LIN {X -0.200,Y -532.074,Z 1046.256,A 0.000,B 0.000,C 90.000,E1 262.129} C_DIS
LIN {X -0.087,Y -530.457,Z 1046.248,A 0.000,B 0.000,C 90.000,E1 260.679} C_DIS
LIN {X 0.126,Y -528.622,Z 1046.239,A 0.000,B 0.000,C 90.000,E1 258.926} C_DIS
LIN {X 0.276,Y -527.082,Z 1046.231,A 0.000,B 0.000,C 90.000,E1 257.465} C_DIS
LIN {X 0.047,Y -524.579,Z 1046.218,A 0.000,B 0.000,C 90.000,E1 255.172} C_DIS
LIN {X 0.007,Y -522.754,Z 1046.208,A 0.000,B 0.000,C 90.000,E1 253.433} C_DIS
LIN {X -0.210,Y -521.218,Z 1046.200,A 0.000,B 0.000,C 90.000,E1 252.000} C_DIS
LIN {X 0.188,Y -519.499,Z 1046.192,A 0.000,B 0.000,C 90.000,E1 250.496} C_DIS
LIN {X 0.026,Y -516.944,Z 1046.180,A 0.000,B 0.000,C 90.000,E1 248.465} C_DIS
LIN {X 0.090,Y -515.507,Z 1046.174,A 0.000,B 0.000,C 90.000,E1 247.283} C_DIS
LIN {X 0.257,Y -513.432,Z 1046.166,A 0.000,B 0.000,C 90.000,E1 245.793} C_DIS
LIN {X 0.125,Y -511.151,Z 1046.157,A 0.000,B 0.000,C 90.000,E1 244.332} C_DIS
LIN {X -0.049,Y -508.765,Z 1046.149,A 0.000,B 0.000,C 90.000,E1 242.871} C_DIS
LIN {X 0.003,Y -507.243,Z 1046.144,A 0.000,B 0.000,C 90.000,E1 241.975} C_DIS
LIN {X 0.221,Y -504.607,Z 1046.136,A 0.000,B 0.000,C 90.000,E1 240.461} C_DIS
LIN {X 0.260,Y -501.301,Z 1046.126,A 0.000,B 0.000,C 90.000,E1 238.663} C_DIS
LIN {X -0.205,Y -497.939,Z 1046.116,A 0.000,B 0.000,C 90.000,E1 236.914} C_DIS
LIN {X 0.081,Y -495.545,Z 1046.109,A 0.000,B 0.000,C 90.000,E1 235.674} C_DIS
LIN {X -0.224,Y -492.350,Z 1046.101,A 0.000,B 0.000,C 90.000,E1 234.196} C_DIS
LIN {X 0.097,Y -488.848,Z 1046.093,A 0.000,B 0.000,C 90.000,E1 232.637} C_DIS
LIN {X 0.258,Y -485.274,Z 1046.084,A 0.000,B 0.000,C 90.000,E1 231.090} C_DIS
LIN {X -0.202,Y -481.123,Z 1046.074,A 0.000,B 0.000,C 90.000,E1 229.299} C_DIS
LIN {X 0.022,Y -476.578,Z 1046.062,A 0.000,B 0.000,C 90.000,E1 227.106} C_DIS
LIN {X -0.022,Y -472.784,Z 1046.051,A 0.000,B 0.000,C 90.000,E1 225.243} C_DIS
LIN {X -0.230,Y -469.527,Z 1046.043,A 0.000,B 0.000,C 90.000,E1 223.704} C_DIS
LIN {X 0.180,Y -466.400,Z 1046.034,A 0.000,B 0.000,C 90.000,E1 222.081} C_DIS
LIN {X -0.129,Y -463.145,Z 1046.025,A 0.000,B 0.000,C 90.000,E1 220.539} C_DIS
LIN {X 0.201,Y -459.845,Z 1046.016,A 0.000,B 0.000,C 90.000,E1 218.910} C_DIS
LIN {X 0.010,Y -454.371,Z 1046.002,A 0.000,B 0.000,C 90.000,E1 216.377} C_DIS
LIN {X 0.035,Y -449.739,Z 1045.990,A 0.000,B 0.000,C 90.000,E1 214.119} C_DIS
LIN {X 0.044,Y -446.432,Z 1045.981,A 0.000,B 0.000,C 90.000,E1 212.498} C_DIS
LIN {X -0.006,Y -442.795,Z 1045.972,A 0.000,B 0.000,C 90.000,E1 210.875} C_DIS
LIN {X 0.202,Y -439.874,Z 1045.964,A 0.000,B 0.000,C 90.000,E1 209.539} C_DIS
LIN {X 0.141,Y -436.975,Z 1045.957,A 0.000,B 0.000,C 90.000,E1 208.231} C_DIS
LIN {X -0.139,Y -432.660,Z 1045.946,A 0.000,B 0.000,C 90.000,E1 206.283} C_DIS
LIN {X 0.031,Y -426.395,Z 1045.929,A 0.000,B 0.000,C 90.000,E1 203.259} C_DIS
LIN {X 0.105,Y -421.444,Z 1045.914,A 0.000,B 0.000,C 90.000,E1 200.556} C_DIS
LIN {X 0.074,Y -416.360,Z 1045.896,A 0.000,B 0.000,C 90.000,E1 197.166} C_DIS
LIN {X -0.051,Y -414.517,Z 1045.884,A 0.000,B 0.000,C 90.000,E1 195.134} C_DIS
LIN {X -0.136,Y -413.982,Z 1045.878,A 0.000,B 0.000,C 90.000,E1 194.120} C_DIS
LIN {X 0.007,Y -413.995,Z 1045.874,A 0.000,B 0.000,C 90.000,E1 193.244} C_DIS
LIN {X 0.114,Y -414.394,Z 1045.871,A 0.000,B 0.000,C 90.000,E1 192.715} C_DIS
LIN {X -0.119,Y -415.327,Z 1045.867,A 0.000,B 0.000,C 90.000,E1 192.063} C_DIS
LIN {X -0.073,Y -416.099,Z 1045.865,A 0.000,B 0.000,C 90.000,E1 191.715} C_DIS
LIN {X 0.043,Y -417.689,Z 1045.862,A 0.000,B 0.000,C 90.000,E1 191.186} C_DIS
LIN {X 0.167,Y -419.693,Z 1045.859,A 0.000,B 0.000,C 90.000,E1 190.658} C_DIS
LIN {X -0.114,Y -423.246,Z 1045.856,A 0.000,B 0.000,C 90.000,E1 190.018} C_DIS
LIN {X 0.049,Y -427.287,Z 1045.852,A 0.000,B 0.000,C 90.000,E1 189.321} C_DIS
LIN {X -0.124,Y -442.017,Z 1045.840,A 0.000,B 0.000,C 90.000,E1 187.182} C_DIS
LIN {X -0.190,Y -447.901,Z 1045.835,A 0.000,B 0.000,C 90.000,E1 186.372} C_DIS
LIN {X 0.121,Y -457.250,Z 1045.828,A 0.000,B 0.000,C 90.000,E1 185.049} C_DIS
LIN {X -0.200,Y -464.000,Z 1045.823,A 0.000,B 0.000,C 90.000,E1 184.131} C_DIS
LIN {X -0.094,Y -469.384,Z 1045.818,A 0.000,B 0.000,C 90.000,E1 183.326} C_DIS
LIN {X 0.062,Y -474.699,Z 1045.814,A 0.000,B 0.000,C 90.000,E1 182.522} C_DIS
LIN {X 0.213,Y -482.614,Z 1045.807,A 0.000,B 0.000,C 90.000,E1 181.260} C_DIS
LIN {X 0.159,Y -488.424,Z 1045.802,A 0.000,B 0.000,C 90.000,E1 180.344} C_DIS
LIN {X 0.170,Y -494.090,Z 1045.797,A 0.000,B 0.000,C 90.000,E1 179.427} C_DIS
LIN {X -0.071,Y -500.502,Z 1045.791,A 0.000,B 0.000,C 90.000,E1 178.396} C_DIS
LIN {X -0.222,Y -506.659,Z 1045.785,A 0.000,B 0.000,C 90.000,E1 177.364} C_DIS
LIN {X -0.212,Y -516.817,Z 1045.775,A 0.000,B 0.000,C 90.000,E1 175.584} C_DIS
LIN {X -0.104,Y -522.664,Z 1045.770,A 0.000,B 0.000,C 90.000,E1 174.546} C_DIS
LIN {X -0.239,Y -530.864,Z 1045.762,A 0.000,B 0.000,C 90.000,E1 173.109} C_DIS
LIN {X -0.101,Y -538.759,Z 1045.754,A 0.000,B 0.000,C 90.000,E1 171.659} C_DIS
LIN {X 0.197,Y -546.551,Z 1045.746,A 0.000,B 0.000,C 90.000,E1 170.208} C_DIS
LIN {X 0.092,Y -554.249,Z 1045.738,A 0.000,B 0.000,C 90.000,E1 168.814} C_DIS
LIN {X -0.184,Y -560.837,Z 1045.731,A 0.000,B 0.000,C 90.000,E1 167.589} C_DIS
LIN {X -0.241,Y -567.323,Z 1045.724,A 0.000,B 0.000,C 90.000,E1 166.353} C_DIS
LIN {X -0.013,Y -570.746,Z 1045.720,A 0.000,B 0.000,C 90.000,E1 165.644} C_DIS
LIN {X -0.218,Y -576.029,Z 1045.714,A 0.000,B 0.000,C 90.000,E1 164.574} C_DIS
LIN {X 0.205,Y -581.233,Z 1045.708,A 0.000,B 0.000,C 90.000,E1 163.449} C_DIS
LIN {X -0.245,Y -586.060,Z 1045.702,A 0.000,B 0.000,C 90.000,E1 162.417} C_DIS
LIN {X 0.066,Y -589.465,Z 1045.698,A 0.000,B 0.000,C 90.000,E1 161.583} C_DIS
LIN {X -0.278,Y -593.772,Z 1045.692,A 0.000,B 0.000,C 90.000,E1 160.550} C_DIS
LIN {X 0.203,Y -597.859,Z 1045.686,A 0.000,B 0.000,C 90.000,E1 159.444} C_DIS
LIN {X 0.056,Y -600.780,Z 1045.682,A 0.000,B 0.000,C 90.000,E1 158.666} C_DIS
LIN {X 0.007,Y -605.255,Z 1045.674,A 0.000,B 0.000,C 90.000,E1 157.358} C_DIS
LIN {X 0.090,Y -608.594,Z 1045.668,A 0.000,B 0.000,C 90.000,E1 156.305} C_DIS
LIN {X -0.127,Y -612.508,Z 1045.661,A 0.000,B 0.000,C 90.000,E1 155.025} C_DIS
LIN {X 0.017,Y -616.093,Z 1045.654,A 0.000,B 0.000,C 90.000,E1 153.717} C_DIS
LIN {X 0.213,Y -619.459,Z 1045.647,A 0.000,B 0.000,C 90.000,E1 152.410} C_DIS
LIN {X 0.185,Y -622.066,Z 1045.641,A 0.000,B 0.000,C 90.000,E1 151.385} C_DIS
LIN {X -0.044,Y -626.476,Z 1045.631,A 0.000,B 0.000,C 90.000,E1 149.616} C_DIS
LIN {X 0.123,Y -630.005,Z 1045.623,A 0.000,B 0.000,C 90.000,E1 148.074} C_DIS
LIN {X 0.324,Y -632.332,Z 1045.617,A 0.000,B 0.000,C 90.000,E1 147.041} C_DIS
LIN {X 0.055,Y -635.173,Z 1045.610,A 0.000,B 0.000,C 90.000,E1 145.801} C_DIS
LIN {X 0.215,Y -638.537,Z 1045.602,A 0.000,B 0.000,C 90.000,E1 144.276} C_DIS
LIN {X -0.106,Y -641.339,Z 1045.595,A 0.000,B 0.000,C 90.000,E1 143.050} C_DIS
LIN {X -0.052,Y -645.284,Z 1045.585,A 0.000,B 0.000,C 90.000,E1 141.295} C_DIS
LIN {X -0.340,Y -648.601,Z 1045.577,A 0.000,B 0.000,C 90.000,E1 139.828} C_DIS
LIN {X -0.154,Y -651.921,Z 1045.568,A 0.000,B 0.000,C 90.000,E1 138.324} C_DIS
LIN {X 0.417,Y -657.092,Z 1045.556,A 0.000,B 0.000,C 90.000,E1 136.053} C_DIS
LIN {X 0.177,Y -664.235,Z 1045.541,A 0.000,B 0.000,C 90.000,E1 133.380} C_DIS
LIN {X 0.181,Y -668.183,Z 1045.533,A 0.000,B 0.000,C 90.000,E1 131.919} C_DIS
LIN {X 0.256,Y -671.593,Z 1045.526,A 0.000,B 0.000,C 90.000,E1 130.701} C_DIS
LIN {X -0.021,Y -676.228,Z 1045.517,A 0.000,B 0.000,C 90.000,E1 129.036} C_DIS
LIN {X -0.277,Y -678.775,Z 1045.512,A 0.000,B 0.000,C 90.000,E1 128.096} C_DIS
LIN {X 0.064,Y -681.852,Z 1045.505,A 0.000,B 0.000,C 90.000,E1 126.870} C_DIS
LIN {X -0.307,Y -686.102,Z 1045.496,A 0.000,B 0.000,C 90.000,E1 125.231} C_DIS
LIN {X -0.417,Y -690.339,Z 1045.486,A 0.000,B 0.000,C 90.000,E1 123.579} C_DIS
LIN {X 0.276,Y -693.178,Z 1045.480,A 0.000,B 0.000,C 90.000,E1 122.339} C_DIS
LIN {X 0.049,Y -695.917,Z 1045.473,A 0.000,B 0.000,C 90.000,E1 121.180} C_DIS
LIN {X 0.194,Y -697.440,Z 1045.469,A 0.000,B 0.000,C 90.000,E1 120.463} C_DIS
LIN {X 0.015,Y -699.086,Z 1045.464,A 0.000,B 0.000,C 90.000,E1 119.539} C_DIS
LIN {X 0.200,Y -700.101,Z 1045.460,A 0.000,B 0.000,C 90.000,E1 118.821} C_DIS
LIN {X -0.024,Y -701.693,Z 1045.453,A 0.000,B 0.000,C 90.000,E1 117.436} C_DIS
LIN {X -0.209,Y -702.998,Z 1045.446,A 0.000,B 0.000,C 90.000,E1 116.283} C_DIS
LIN {X -0.024,Y -703.814,Z 1045.441,A 0.000,B 0.000,C 90.000,E1 115.335} C_DIS
LIN {X -0.109,Y -704.204,Z 1045.437,A 0.000,B 0.000,C 90.000,E1 114.643} C_DIS
LIN {X 0.168,Y -704.031,Z 1045.434,A 0.000,B 0.000,C 90.000,E1 114.155} C_DIS
LIN {X -0.190,Y -703.680,Z 1045.433,A 0.000,B 0.000,C 90.000,E1 113.951} C_DIS
LIN {X 0.089,Y -702.567,Z 1045.430,A 0.000,B 0.000,C 90.000,E1 113.462} C_DIS
LIN {X -0.278,Y -701.385,Z 1045.429,A 0.000,B 0.000,C 90.000,E1 113.259} C_DIS
LIN {X -0.011,Y -698.386,Z 1045.427,A 0.000,B 0.000,C 90.000,E1 112.770} C_DIS
LIN {X 0.120,Y -697.192,Z 1045.426,A 0.000,B 0.000,C 90.000,E1 112.642} C_DIS
LIN {X 0.249,Y -695.337,Z 1045.425,A 0.000,B 0.000,C 90.000,E1 112.514} C_DIS
LIN {X -0.172,Y -688.457,Z 1045.423,A 0.000,B 0.000,C 90.000,E1 112.206} C_DIS
LIN {X 0.181,Y -686.259,Z 1045.423,A 0.000,B 0.000,C 90.000,E1 112.099} C_DIS
LIN {X 0.154,Y -682.920,Z 1045.422,A 0.000,B 0.000,C 90.000,E1 112.025} C_DIS
LIN {X 0.001,Y -675.996,Z 1045.422,A 0.000,B 0.000,C 90.000,E1 111.950} C_DIS
LIN {X -0.058,Y -610.637,Z 1045.422,A 0.000,B 0.000,C 90.000,E1 111.950} C_DIS
LIN {X 0.150,Y -604.476,Z 1045.421,A 0.000,B 0.000,C 90.000,E1 111.716} C_DIS
LIN {X 0.007,Y -598.087,Z 1045.419,A 0.000,B 0.000,C 90.000,E1 111.408} C_DIS
LIN {X -0.080,Y -592.488,Z 1045.417,A 0.000,B 0.000,C 90.000,E1 111.046} C_DIS
LIN {X -0.061,Y -576.610,Z 1045.410,A 0.000,B 0.000,C 90.000,E1 109.758} C_DIS
LIN {X 0.286,Y -570.579,Z 1045.407,A 0.000,B 0.000,C 90.000,E1 109.268} C_DIS
LIN {X -0.275,Y -568.981,Z 1045.407,A 0.000,B 0.000,C 90.000,E1 109.214} C_DIS
LIN {X -0.188,Y -560.664,Z 1045.404,A 0.000,B 0.000,C 90.000,E1 108.725} C_DIS
LIN {X -0.120,Y -554.210,Z 1045.402,A 0.000,B 0.000,C 90.000,E1 108.362} C_DIS
LIN {X 0.095,Y -549.849,Z 1045.400,A 0.000,B 0.000,C 90.000,E1 108.055} C_DIS
LIN {X 0.152,Y -548.856,Z 1045.400,A 0.000,B 0.000,C 90.000,E1 107.946} C_DIS
LIN {X 0.230,Y -547.887,Z 1045.399,A 0.000,B 0.000,C 90.000,E1 107.819} C_DIS
LIN {X 0.188,Y -547.874,Z 1045.399,A 0.000,B 0.000,C 90.000,E1 107.819} C_DIS
LIN {X 0.273,Y -547.436,Z 1045.397,A 0.000,B 0.000,C 90.000,E1 107.511} C_DIS
LIN {X -0.215,Y -547.637,Z 1045.394,A 0.000,B 0.000,C 90.000,E1 106.858} C_DIS
LIN {X -0.069,Y -548.307,Z 1045.387,A 0.000,B 0.000,C 90.000,E1 105.717} C_DIS
LIN {X 0.139,Y -549.314,Z 1045.378,A 0.000,B 0.000,C 90.000,E1 104.008} C_DIS
LIN {X -0.248,Y -551.520,Z 1045.362,A 0.000,B 0.000,C 90.000,E1 101.243} C_DIS
LIN {X 0.091,Y -554.167,Z 1045.348,A 0.000,B 0.000,C 90.000,E1 98.690} C_DIS
LIN {X 0.263,Y -556.428,Z 1045.338,A 0.000,B 0.000,C 90.000,E1 96.720} C_DIS
LIN {X 0.021,Y -557.372,Z 1045.333,A 0.000,B 0.000,C 90.000,E1 95.910} C_DIS
LIN {X -0.073,Y -558.612,Z 1045.325,A 0.000,B 0.000,C 90.000,E1 94.531} C_DIS
LIN {X 0.209,Y -559.234,Z 1045.321,A 0.000,B 0.000,C 90.000,E1 93.669} C_DIS
LIN {X 0.117,Y -560.028,Z 1045.313,A 0.000,B 0.000,C 90.000,E1 92.293} C_DIS
LIN {X -0.057,Y -560.523,Z 1045.307,A 0.000,B 0.000,C 90.000,E1 91.203} C_DIS
LIN {X -0.047,Y -561.123,Z 1045.297,A 0.000,B 0.000,C 90.000,E1 89.542} C_DIS
LIN {X 0.087,Y -561.716,Z 1045.287,A 0.000,B 0.000,C 90.000,E1 87.593} C_DIS
LIN {X 0.262,Y -562.424,Z 1045.276,A 0.000,B 0.000,C 90.000,E1 85.641} C_DIS
LIN {X 0.259,Y -562.824,Z 1045.268,A 0.000,B 0.000,C 90.000,E1 84.261} C_DIS
LIN {X -0.154,Y -563.234,Z 1045.259,A 0.000,B 0.000,C 90.000,E1 82.648} C_DIS
LIN {X -0.008,Y -563.977,Z 1045.245,A 0.000,B 0.000,C 90.000,E1 80.151} C_DIS
LIN {X 0.262,Y -565.056,Z 1045.232,A 0.000,B 0.000,C 90.000,E1 77.645} C_DIS
LIN {X 0.082,Y -566.274,Z 1045.219,A 0.000,B 0.000,C 90.000,E1 75.463} C_DIS
LIN {X -0.138,Y -568.069,Z 1045.206,A 0.000,B 0.000,C 90.000,E1 73.015} C_DIS
LIN {X 0.099,Y -569.400,Z 1045.197,A 0.000,B 0.000,C 90.000,E1 71.348} C_DIS
LIN {X -0.169,Y -570.571,Z 1045.189,A 0.000,B 0.000,C 90.000,E1 70.007} C_DIS
LIN {X -0.032,Y -571.345,Z 1045.183,A 0.000,B 0.000,C 90.000,E1 68.901} C_DIS
LIN {X -0.054,Y -572.361,Z 1045.175,A 0.000,B 0.000,C 90.000,E1 67.539} C_DIS
LIN {X 0.135,Y -573.580,Z 1045.165,A 0.000,B 0.000,C 90.000,E1 65.613} C_DIS
LIN {X -0.302,Y -574.435,Z 1045.156,A 0.000,B 0.000,C 90.000,E1 64.024} C_DIS
LIN {X 0.048,Y -575.261,Z 1045.146,A 0.000,B 0.000,C 90.000,E1 62.359} C_DIS
LIN {X 0.024,Y -576.087,Z 1045.136,A 0.000,B 0.000,C 90.000,E1 60.461} C_DIS
LIN {X -0.329,Y -576.869,Z 1045.127,A 0.000,B 0.000,C 90.000,E1 58.869} C_DIS
LIN {X 0.117,Y -577.427,Z 1045.118,A 0.000,B 0.000,C 90.000,E1 57.199} C_DIS
LIN {X -0.239,Y -577.784,Z 1045.110,A 0.000,B 0.000,C 90.000,E1 55.881} C_DIS
LIN {X 0.220,Y -578.048,Z 1045.103,A 0.000,B 0.000,C 90.000,E1 54.482} C_DIS
LIN {X 0.054,Y -578.175,Z 1045.097,A 0.000,B 0.000,C 90.000,E1 53.417} C_DIS
LIN {X -0.114,Y -578.127,Z 1045.091,A 0.000,B 0.000,C 90.000,E1 52.351} C_DIS
LIN {X 0.070,Y -577.884,Z 1045.085,A 0.000,B 0.000,C 90.000,E1 51.251} C_DIS
LIN {X -0.040,Y -577.314,Z 1045.077,A 0.000,B 0.000,C 90.000,E1 49.908} C_DIS
LIN {X -0.162,Y -576.592,Z 1045.070,A 0.000,B 0.000,C 90.000,E1 48.566} C_DIS
LIN {X -0.063,Y -575.880,Z 1045.064,A 0.000,B 0.000,C 90.000,E1 47.472} C_DIS
LIN {X 0.029,Y -575.014,Z 1045.058,A 0.000,B 0.000,C 90.000,E1 46.377} C_DIS
LIN {X -0.306,Y -573.795,Z 1045.052,A 0.000,B 0.000,C 90.000,E1 45.324} C_DIS
LIN {X 0.039,Y -572.701,Z 1045.047,A 0.000,B 0.000,C 90.000,E1 44.474} C_DIS
LIN {X 0.079,Y -571.027,Z 1045.041,A 0.000,B 0.000,C 90.000,E1 43.380} C_DIS
LIN {X 0.017,Y -569.627,Z 1045.036,A 0.000,B 0.000,C 90.000,E1 42.567} C_DIS
LIN {X -0.092,Y -568.048,Z 1045.032,A 0.000,B 0.000,C 90.000,E1 41.757} C_DIS
LIN {X 0.198,Y -566.255,Z 1045.027,A 0.000,B 0.000,C 90.000,E1 40.906} C_DIS
LIN {X -0.011,Y -565.016,Z 1045.024,A 0.000,B 0.000,C 90.000,E1 40.378} C_DIS
LIN {X -0.122,Y -562.791,Z 1045.020,A 0.000,B 0.000,C 90.000,E1 39.564} C_DIS
LIN {X 0.083,Y -561.274,Z 1045.017,A 0.000,B 0.000,C 90.000,E1 38.991} C_DIS
LIN {X -0.064,Y -558.586,Z 1045.012,A 0.000,B 0.000,C 90.000,E1 38.177} C_DIS
LIN {X -0.162,Y -554.661,Z 1045.006,A 0.000,B 0.000,C 90.000,E1 37.076} C_DIS
LIN {X -0.013,Y -552.442,Z 1045.003,A 0.000,B 0.000,C 90.000,E1 36.503} C_DIS
LIN {X -0.143,Y -548.738,Z 1044.998,A 0.000,B 0.000,C 90.000,E1 35.678} C_DIS
LIN {X -0.133,Y -544.187,Z 1044.993,A 0.000,B 0.000,C 90.000,E1 34.692} C_DIS
LIN {X -0.046,Y -539.818,Z 1044.988,A 0.000,B 0.000,C 90.000,E1 33.833} C_DIS
LIN {X -0.006,Y -534.438,Z 1044.982,A 0.000,B 0.000,C 90.000,E1 32.832} C_DIS
LIN {X 0.100,Y -527.592,Z 1044.976,A 0.000,B 0.000,C 90.000,E1 31.671} C_DIS
LIN {X -0.247,Y -523.884,Z 1044.973,A 0.000,B 0.000,C 90.000,E1 31.131} C_DIS
LIN {X -0.071,Y -518.983,Z 1044.969,A 0.000,B 0.000,C 90.000,E1 30.384} C_DIS
LIN {X -0.033,Y -514.771,Z 1044.966,A 0.000,B 0.000,C 90.000,E1 29.795} C_DIS
LIN {X 0.152,Y -511.416,Z 1044.963,A 0.000,B 0.000,C 90.000,E1 29.333} C_DIS
LIN {X 0.021,Y -504.457,Z 1044.958,A 0.000,B 0.000,C 90.000,E1 28.487} C_DIS
LIN {X 0.020,Y -499.282,Z 1044.955,A 0.000,B 0.000,C 90.000,E1 27.897} C_DIS
LIN {X 0.238,Y -491.048,Z 1044.950,A 0.000,B 0.000,C 90.000,E1 27.001} C_DIS
LIN {X 0.081,Y -484.067,Z 1044.946,A 0.000,B 0.000,C 90.000,E1 26.309} C_DIS
LIN {X 0.103,Y -474.008,Z 1044.941,A 0.000,B 0.000,C 90.000,E1 25.335} C_DIS
LIN {X 0.155,Y -463.659,Z 1044.936,A 0.000,B 0.000,C 90.000,E1 24.387} C_DIS
LIN {X -0.078,Y -453.086,Z 1044.931,A 0.000,B 0.000,C 90.000,E1 23.515} C_DIS
LIN {X 0.100,Y -429.481,Z 1044.919,A 0.000,B 0.000,C 90.000,E1 21.408} C_DIS
LIN {X -0.117,Y -417.985,Z 1044.913,A 0.000,B 0.000,C 90.000,E1 20.301} C_DIS
LIN {X -0.190,Y -406.782,Z 1044.906,A 0.000,B 0.000,C 90.000,E1 19.087} C_DIS
LIN {X -0.056,Y -400.031,Z 1044.901,A 0.000,B 0.000,C 90.000,E1 18.236} C_DIS
LIN {X 0.082,Y -396.246,Z 1044.898,A 0.000,B 0.000,C 90.000,E1 17.692} C_DIS
LIN {X 0.117,Y -395.210,Z 1044.897,A 0.000,B 0.000,C 90.000,E1 17.511} C_DIS
LIN {X -0.148,Y -392.499,Z 1044.894,A 0.000,B 0.000,C 90.000,E1 16.913} C_DIS
LIN {X -0.073,Y -391.496,Z 1044.891,A 0.000,B 0.000,C 90.000,E1 16.370} C_DIS
LIN {X 0.141,Y -391.410,Z 1044.887,A 0.000,B 0.000,C 90.000,E1 15.717} C_DIS
LIN {X 0.067,Y -392.262,Z 1044.882,A 0.000,B 0.000,C 90.000,E1 14.662} C_DIS
LIN {X -0.027,Y -398.877,Z 1044.854,A 0.000,B 0.000,C 90.000,E1 9.726} C_DIS
LIN {X 0.163,Y -406.120,Z 1044.833,A 0.000,B 0.000,C 90.000,E1 5.853} C_DIS
LIN {X 0.113,Y -409.107,Z 1044.825,A 0.000,B 0.000,C 90.000,E1 4.473} C_DIS
LIN {X 0.091,Y -411.905,Z 1044.818,A 0.000,B 0.000,C 90.000,E1 3.269} C_DIS
LIN {X 0.107,Y -413.904,Z 1044.815,A 0.000,B 0.000,C 90.000,E1 2.751} C_DIS
LIN {X 0.198,Y -414.700,Z 1044.815,A 0.000,B 0.000,C 90.000,E1 2.579} C_DIS
LIN {X -0.114,Y -418.010,Z 1044.812,A 0.000,B 0.000,C 90.000,E1 2.121} C_DIS
LIN {X 0.084,Y -421.155,Z 1044.810,A 0.000,B 0.000,C 90.000,E1 1.776} C_DIS
LIN {X -0.058,Y -422.789,Z 1044.809,A 0.000,B 0.000,C 90.000,E1 1.661} C_DIS
LIN {X -0.160,Y -436.414,Z 1044.804,A 0.000,B 0.000,C 90.000,E1 0.802} C_DIS
LIN {X -0.182,Y -453.799,Z 1044.798,A 0.000,B 0.000,C 90.000,E1 359.714} C_DIS
LIN {X 0.113,Y -472.035,Z 1044.792,A 0.000,B 0.000,C 90.000,E1 358.568} C_DIS
LIN {X -0.212,Y -486.861,Z 1044.787,A 0.000,B 0.000,C 90.000,E1 357.707} C_DIS
LIN {X 0.018,Y -496.616,Z 1044.784,A 0.000,B 0.000,C 90.000,E1 357.078} C_DIS
LIN {X -0.004,Y -504.469,Z 1044.781,A 0.000,B 0.000,C 90.000,E1 356.560} C_DIS
LIN {X 0.215,Y -510.656,Z 1044.779,A 0.000,B 0.000,C 90.000,E1 356.102} C_DIS
LIN {X -0.040,Y -516.687,Z 1044.776,A 0.000,B 0.000,C 90.000,E1 355.698} C_DIS
LIN {X -0.028,Y -525.260,Z 1044.772,A 0.000,B 0.000,C 90.000,E1 355.008} C_DIS
LIN {X 0.107,Y -532.364,Z 1044.769,A 0.000,B 0.000,C 90.000,E1 354.375} C_DIS
LIN {X -0.068,Y -539.086,Z 1044.765,A 0.000,B 0.000,C 90.000,E1 353.742} C_DIS
LIN {X 0.038,Y -545.438,Z 1044.761,A 0.000,B 0.000,C 90.000,E1 353.053} C_DIS
LIN {X 0.263,Y -550.224,Z 1044.758,A 0.000,B 0.000,C 90.000,E1 352.470} C_DIS
LIN {X -0.141,Y -554.661,Z 1044.755,A 0.000,B 0.000,C 90.000,E1 351.951} C_DIS
LIN {X -0.140,Y -559.523,Z 1044.751,A 0.000,B 0.000,C 90.000,E1 351.254} C_DIS
LIN {X -0.092,Y -563.883,Z 1044.748,A 0.000,B 0.000,C 90.000,E1 350.557} C_DIS
LIN {X -0.249,Y -568.647,Z 1044.743,A 0.000,B 0.000,C 90.000,E1 349.746} C_DIS
LIN {X 0.307,Y -573.054,Z 1044.738,A 0.000,B 0.000,C 90.000,E1 348.870} C_DIS
LIN {X -0.213,Y -577.031,Z 1044.734,A 0.000,B 0.000,C 90.000,E1 348.105} C_DIS
LIN {X -0.018,Y -580.092,Z 1044.730,A 0.000,B 0.000,C 90.000,E1 347.409} C_DIS
LIN {X -0.245,Y -584.740,Z 1044.724,A 0.000,B 0.000,C 90.000,E1 346.353} C_DIS
LIN {X -0.195,Y -586.901,Z 1044.721,A 0.000,B 0.000,C 90.000,E1 345.811} C_DIS
LIN {X -0.230,Y -593.200,Z 1044.712,A 0.000,B 0.000,C 90.000,E1 344.212} C_DIS
LIN {X -0.133,Y -597.210,Z 1044.706,A 0.000,B 0.000,C 90.000,E1 343.142} C_DIS
LIN {X -0.270,Y -600.019,Z 1044.702,A 0.000,B 0.000,C 90.000,E1 342.362} C_DIS
LIN {X -0.185,Y -604.459,Z 1044.695,A 0.000,B 0.000,C 90.000,E1 341.040} C_DIS
LIN {X -0.331,Y -607.595,Z 1044.689,A 0.000,B 0.000,C 90.000,E1 340.007} C_DIS
LIN {X -0.164,Y -609.914,Z 1044.684,A 0.000,B 0.000,C 90.000,E1 339.209} C_DIS
LIN {X 0.028,Y -611.979,Z 1044.680,A 0.000,B 0.000,C 90.000,E1 338.411} C_DIS
LIN {X 0.173,Y -615.272,Z 1044.673,A 0.000,B 0.000,C 90.000,E1 337.102} C_DIS
LIN {X -0.186,Y -618.259,Z 1044.666,A 0.000,B 0.000,C 90.000,E1 335.845} C_DIS
LIN {X 0.062,Y -620.816,Z 1044.659,A 0.000,B 0.000,C 90.000,E1 334.537} C_DIS
LIN {X 0.052,Y -622.599,Z 1044.653,A 0.000,B 0.000,C 90.000,E1 333.512} C_DIS
LIN {X 0.066,Y -624.247,Z 1044.647,A 0.000,B 0.000,C 90.000,E1 332.487} C_DIS
LIN {X 0.096,Y -625.731,Z 1044.642,A 0.000,B 0.000,C 90.000,E1 331.463} C_DIS
LIN {X -0.092,Y -627.317,Z 1044.635,A 0.000,B 0.000,C 90.000,E1 330.205} C_DIS
LIN {X 0.086,Y -628.782,Z 1044.626,A 0.000,B 0.000,C 90.000,E1 328.663} C_DIS
LIN {X -0.067,Y -629.591,Z 1044.620,A 0.000,B 0.000,C 90.000,E1 327.661} C_DIS
LIN {X -0.035,Y -630.303,Z 1044.612,A 0.000,B 0.000,C 90.000,E1 326.135} C_DIS
LIN {X 0.172,Y -630.499,Z 1044.606,A 0.000,B 0.000,C 90.000,E1 325.102} C_DIS
LIN {X -0.292,Y -630.575,Z 1044.598,A 0.000,B 0.000,C 90.000,E1 323.623} C_DIS
LIN {X 0.343,Y -630.566,Z 1044.587,A 0.000,B 0.000,C 90.000,E1 321.537} C_DIS
LIN {X -0.079,Y -630.692,Z 1044.581,A 0.000,B 0.000,C 90.000,E1 320.561} C_DIS
LIN {X 0.219,Y -630.855,Z 1044.573,A 0.000,B 0.000,C 90.000,E1 319.013} C_DIS
LIN {X -0.017,Y -630.814,Z 1044.564,A 0.000,B 0.000,C 90.000,E1 317.514} C_DIS
LIN {X 0.103,Y -631.007,Z 1044.554,A 0.000,B 0.000,C 90.000,E1 315.729} C_DIS
LIN {X 0.204,Y -631.189,Z 1044.544,A 0.000,B 0.000,C 90.000,E1 313.947} C_DIS
LIN {X -0.137,Y -631.350,Z 1044.534,A 0.000,B 0.000,C 90.000,E1 312.204} C_DIS
LIN {X -0.315,Y -631.315,Z 1044.526,A 0.000,B 0.000,C 90.000,E1 310.701} C_DIS
LIN {X 0.164,Y -631.342,Z 1044.520,A 0.000,B 0.000,C 90.000,E1 309.644} C_DIS
LIN {X -0.251,Y -631.259,Z 1044.515,A 0.000,B 0.000,C 90.000,E1 308.669} C_DIS
LIN {X 0.031,Y -631.204,Z 1044.505,A 0.000,B 0.000,C 90.000,E1 306.870} C_DIS
LIN {X -0.122,Y -631.192,Z 1044.502,A 0.000,B 0.000,C 90.000,E1 306.377} C_DIS
LIN {X 0.244,Y -631.294,Z 1044.501,A 0.000,B 0.000,C 90.000,E1 306.091} C_DIS
LIN {X -0.124,Y -632.078,Z 1044.482,A 0.000,B 0.000,C 90.000,E1 302.832} C_DIS
LIN {X -0.030,Y -632.871,Z 1044.473,A 0.000,B 0.000,C 90.000,E1 301.052} C_DIS
LIN {X 0.012,Y -634.193,Z 1044.461,A 0.000,B 0.000,C 90.000,E1 299.027} C_DIS
LIN {X -0.035,Y -635.105,Z 1044.454,A 0.000,B 0.000,C 90.000,E1 297.769} C_DIS
LIN {X 0.146,Y -635.734,Z 1044.449,A 0.000,B 0.000,C 90.000,E1 296.744} C_DIS
LIN {X 0.288,Y -636.117,Z 1044.444,A 0.000,B 0.000,C 90.000,E1 295.976} C_DIS
LIN {X -0.318,Y -636.187,Z 1044.438,A 0.000,B 0.000,C 90.000,E1 294.771} C_DIS
LIN {X -0.392,Y -635.957,Z 1044.432,A 0.000,B 0.000,C 90.000,E1 293.770} C_DIS
LIN {X 0.197,Y -635.086,Z 1044.423,A 0.000,B 0.000,C 90.000,E1 292.206} C_DIS
LIN {X -0.004,Y -634.887,Z 1044.422,A 0.000,B 0.000,C 90.000,E1 291.972} C_DIS
LIN {X 0.065,Y -634.107,Z 1044.419,A 0.000,B 0.000,C 90.000,E1 291.461} C_DIS
LIN {X -0.134,Y -633.676,Z 1044.418,A 0.000,B 0.000,C 90.000,E1 291.227} C_DIS
LIN {X -0.304,Y -632.059,Z 1044.415,A 0.000,B 0.000,C 90.000,E1 290.737} C_DIS
LIN {X -0.280,Y -630.964,Z 1044.414,A 0.000,B 0.000,C 90.000,E1 290.482} C_DIS
LIN {X 0.122,Y -628.028,Z 1044.411,A 0.000,B 0.000,C 90.000,E1 289.939} C_DIS
LIN {X -0.032,Y -623.121,Z 1044.408,A 0.000,B 0.000,C 90.000,E1 289.450} C_DIS
LIN {X 0.011,Y -621.560,Z 1044.407,A 0.000,B 0.000,C 90.000,E1 289.322} C_DIS
LIN {X 0.138,Y -615.029,Z 1044.405,A 0.000,B 0.000,C 90.000,E1 288.906} C_DIS
LIN {X -0.091,Y -613.041,Z 1044.405,A 0.000,B 0.000,C 90.000,E1 288.833} C_DIS
LIN {X 0.046,Y -607.375,Z 1044.403,A 0.000,B 0.000,C 90.000,E1 288.598} C_DIS
LIN {X 0.191,Y -603.694,Z 1044.402,A 0.000,B 0.000,C 90.000,E1 288.417} C_DIS
LIN {X -0.107,Y -597.924,Z 1044.401,A 0.000,B 0.000,C 90.000,E1 288.236} C_DIS
LIN {X -0.192,Y -594.648,Z 1044.401,A 0.000,B 0.000,C 90.000,E1 288.109} C_DIS
LIN {X -0.226,Y -585.329,Z 1044.399,A 0.000,B 0.000,C 90.000,E1 287.819} C_DIS
LIN {X -0.271,Y -578.675,Z 1044.398,A 0.000,B 0.000,C 90.000,E1 287.638} C_DIS
LIN {X 0.227,Y -566.900,Z 1044.396,A 0.000,B 0.000,C 90.000,E1 287.221} C_DIS
LIN {X 0.213,Y -558.710,Z 1044.394,A 0.000,B 0.000,C 90.000,E1 286.913} C_DIS
LIN {X 0.090,Y -553.768,Z 1044.393,A 0.000,B 0.000,C 90.000,E1 286.677} C_DIS
LIN {X 0.200,Y -552.023,Z 1044.392,A 0.000,B 0.000,C 90.000,E1 286.567} C_DIS
LIN {X 0.039,Y -550.106,Z 1044.391,A 0.000,B 0.000,C 90.000,E1 286.315} C_DIS
LIN {X -0.221,Y -549.058,Z 1044.389,A 0.000,B 0.000,C 90.000,E1 286.024} C_DIS
LIN {X -0.156,Y -548.237,Z 1044.386,A 0.000,B 0.000,C 90.000,E1 285.426} C_DIS
LIN {X 0.281,Y -547.552,Z 1044.381,A 0.000,B 0.000,C 90.000,E1 284.537} C_DIS
LIN {X 0.031,Y -547.134,Z 1044.376,A 0.000,B 0.000,C 90.000,E1 283.592} C_DIS
LIN {X 0.000,Y -547.134,Z 1044.376,A 0.000,B 0.000,C 90.000,E1 283.592} C_DIS
LIN {X -0.052,Y -547.497,Z 1044.375,A 0.000,B 0.000,C 90.000,E1 283.536} C_DIS
LIN {X -0.093,Y -585.817,Z 1044.375,A 0.000,B 0.000,C 90.000,E1 283.536} C_DIS
LIN {X 0.293,Y -587.216,Z 1044.375,A 0.000,B 0.000,C 90.000,E1 283.411} C_DIS
LIN {X 0.022,Y -589.821,Z 1044.374,A 0.000,B 0.000,C 90.000,E1 283.244} C_DIS
LIN {X 0.212,Y -592.128,Z 1044.372,A 0.000,B 0.000,C 90.000,E1 283.008} C_DIS
LIN {X 0.074,Y -592.701,Z 1044.371,A 0.000,B 0.000,C 90.000,E1 282.771} C_DIS
LIN {X 0.043,Y -592.729,Z 1044.368,A 0.000,B 0.000,C 90.000,E1 282.243} C_DIS
LIN {X 0.015,Y -591.728,Z 1044.365,A 0.000,B 0.000,C 90.000,E1 281.715} C_DIS
LIN {X -0.233,Y -589.460,Z 1044.361,A 0.000,B 0.000,C 90.000,E1 281.074} C_DIS
LIN {X -0.071,Y -586.865,Z 1044.359,A 0.000,B 0.000,C 90.000,E1 280.658} C_DIS
LIN {X -0.286,Y -585.571,Z 1044.359,A 0.000,B 0.000,C 90.000,E1 280.546} C_DIS
LIN {X 0.182,Y -583.744,Z 1044.358,A 0.000,B 0.000,C 90.000,E1 280.366} C_DIS
LIN {X -0.297,Y -581.323,Z 1044.357,A 0.000,B 0.000,C 90.000,E1 280.197} C_DIS
LIN {X -0.199,Y -580.267,Z 1044.356,A 0.000,B 0.000,C 90.000,E1 280.074} C_DIS
LIN {X -0.282,Y -578.638,Z 1044.355,A 0.000,B 0.000,C 90.000,E1 279.962} C_DIS
LIN {X 0.249,Y -578.442,Z 1044.355,A 0.000,B 0.000,C 90.000,E1 279.905} C_DIS
LIN {X 0.209,Y -572.472,Z 1044.355,A 0.000,B 0.000,C 90.000,E1 279.905} C_DIS
LIN {X 0.158,Y -572.093,Z 1044.355,A 0.000,B 0.000,C 90.000,E1 279.905} C_DIS
LIN {X 0.103,Y -544.908,Z 1044.355,A 0.000,B 0.000,C 90.000,E1 279.905} C_DIS
LIN {X -0.242,Y -543.004,Z 1044.343,A 0.000,B 0.000,C 90.000,E1 277.757} C_DIS
LIN {X 0.096,Y -541.398,Z 1044.330,A 0.000,B 0.000,C 90.000,E1 275.454} C_DIS
LIN {X -0.204,Y -540.168,Z 1044.319,A 0.000,B 0.000,C 90.000,E1 273.498} C_DIS
LIN {X -0.043,Y -539.041,Z 1044.308,A 0.000,B 0.000,C 90.000,E1 271.489} C_DIS
LIN {X 0.017,Y -538.376,Z 1044.302,A 0.000,B 0.000,C 90.000,E1 270.344} C_DIS
LIN {X 0.090,Y -537.262,Z 1044.292,A 0.000,B 0.000,C 90.000,E1 268.625} C_DIS
LIN {X 0.140,Y -536.257,Z 1044.285,A 0.000,B 0.000,C 90.000,E1 267.192} C_DIS
LIN {X 0.173,Y -535.448,Z 1044.278,A 0.000,B 0.000,C 90.000,E1 266.045} C_DIS
LIN {X 0.244,Y -534.002,Z 1044.267,A 0.000,B 0.000,C 90.000,E1 264.033} C_DIS
LIN {X -0.209,Y -532.825,Z 1044.259,A 0.000,B 0.000,C 90.000,E1 262.648} C_DIS
LIN {X -0.080,Y -531.273,Z 1044.251,A 0.000,B 0.000,C 90.000,E1 261.197} C_DIS
LIN {X 0.127,Y -528.746,Z 1044.238,A 0.000,B 0.000,C 90.000,E1 258.870} C_DIS
LIN {X -0.237,Y -527.209,Z 1044.230,A 0.000,B 0.000,C 90.000,E1 257.465} C_DIS
LIN {X 0.180,Y -524.703,Z 1044.217,A 0.000,B 0.000,C 90.000,E1 255.102} C_DIS
LIN {X 0.004,Y -522.871,Z 1044.208,A 0.000,B 0.000,C 90.000,E1 253.378} C_DIS
LIN {X -0.215,Y -521.332,Z 1044.200,A 0.000,B 0.000,C 90.000,E1 251.945} C_DIS
LIN {X -0.135,Y -519.592,Z 1044.192,A 0.000,B 0.000,C 90.000,E1 250.477} C_DIS
LIN {X 0.016,Y -517.044,Z 1044.180,A 0.000,B 0.000,C 90.000,E1 248.411} C_DIS
LIN {X 0.078,Y -515.613,Z 1044.174,A 0.000,B 0.000,C 90.000,E1 247.230} C_DIS
LIN {X -0.228,Y -513.529,Z 1044.165,A 0.000,B 0.000,C 90.000,E1 245.793} C_DIS
LIN {X 0.105,Y -511.237,Z 1044.157,A 0.000,B 0.000,C 90.000,E1 244.280} C_DIS
LIN {X -0.169,Y -509.341,Z 1044.151,A 0.000,B 0.000,C 90.000,E1 243.127} C_DIS
LIN {X -0.108,Y -507.878,Z 1044.146,A 0.000,B 0.000,C 90.000,E1 242.231} C_DIS
LIN {X -0.249,Y -504.666,Z 1044.136,A 0.000,B 0.000,C 90.000,E1 240.461} C_DIS
LIN {X -0.080,Y -501.940,Z 1044.127,A 0.000,B 0.000,C 90.000,E1 238.948} C_DIS
LIN {X 0.155,Y -498.584,Z 1044.117,A 0.000,B 0.000,C 90.000,E1 237.120} C_DIS
LIN {X 0.038,Y -496.223,Z 1044.111,A 0.000,B 0.000,C 90.000,E1 235.928} C_DIS
LIN {X 0.035,Y -494.301,Z 1044.106,A 0.000,B 0.000,C 90.000,E1 235.022} C_DIS
LIN {X 0.009,Y -492.349,Z 1044.101,A 0.000,B 0.000,C 90.000,E1 234.116} C_DIS
LIN {X -0.057,Y -488.832,Z 1044.092,A 0.000,B 0.000,C 90.000,E1 232.603} C_DIS
LIN {X -0.020,Y -485.988,Z 1044.085,A 0.000,B 0.000,C 90.000,E1 231.376} C_DIS
LIN {X -0.094,Y -481.792,Z 1044.075,A 0.000,B 0.000,C 90.000,E1 229.542} C_DIS
LIN {X -0.206,Y -477.221,Z 1044.063,A 0.000,B 0.000,C 90.000,E1 227.391} C_DIS
LIN {X 0.111,Y -473.413,Z 1044.053,A 0.000,B 0.000,C 90.000,E1 225.486} C_DIS
LIN {X -0.086,Y -470.119,Z 1044.044,A 0.000,B 0.000,C 90.000,E1 223.947} C_DIS
LIN {X -0.009,Y -467.006,Z 1044.035,A 0.000,B 0.000,C 90.000,E1 222.366} C_DIS
LIN {X 0.093,Y -463.081,Z 1044.025,A 0.000,B 0.000,C 90.000,E1 220.458} C_DIS
LIN {X -0.227,Y -459.801,Z 1044.016,A 0.000,B 0.000,C 90.000,E1 218.910} C_DIS
LIN {X 0.221,Y -454.253,Z 1044.002,A 0.000,B 0.000,C 90.000,E1 216.297} C_DIS
LIN {X -0.016,Y -449.650,Z 1043.989,A 0.000,B 0.000,C 90.000,E1 214.072} C_DIS
LIN {X -0.138,Y -446.331,Z 1043.980,A 0.000,B 0.000,C 90.000,E1 212.467} C_DIS
LIN {X 0.236,Y -441.945,Z 1043.969,A 0.000,B 0.000,C 90.000,E1 210.463} C_DIS
LIN {X -0.175,Y -439.009,Z 1043.962,A 0.000,B 0.000,C 90.000,E1 209.205} C_DIS
LIN {X 0.108,Y -436.780,Z 1043.957,A 0.000,B 0.000,C 90.000,E1 208.180} C_DIS
LIN {X -0.170,Y -432.438,Z 1043.946,A 0.000,B 0.000,C 90.000,E1 206.232} C_DIS
LIN {X 0.002,Y -426.143,Z 1043.929,A 0.000,B 0.000,C 90.000,E1 203.206} C_DIS
LIN {X 0.045,Y -421.732,Z 1043.916,A 0.000,B 0.000,C 90.000,E1 200.844} C_DIS
LIN {X -0.204,Y -415.533,Z 1043.893,A 0.000,B 0.000,C 90.000,E1 196.804} C_DIS
LIN {X 0.015,Y -413.920,Z 1043.884,A 0.000,B 0.000,C 90.000,E1 195.064} C_DIS
LIN {X -0.181,Y -413.375,Z 1043.878,A 0.000,B 0.000,C 90.000,E1 194.064} C_DIS
LIN {X 0.022,Y -413.139,Z 1043.872,A 0.000,B 0.000,C 90.000,E1 193.008} C_DIS
LIN {X 0.185,Y -413.688,Z 1043.869,A 0.000,B 0.000,C 90.000,E1 192.299} C_DIS
LIN {X -0.140,Y -414.715,Z 1043.865,A 0.000,B 0.000,C 90.000,E1 191.658} C_DIS
LIN {X -0.014,Y -415.545,Z 1043.863,A 0.000,B 0.000,C 90.000,E1 191.299} C_DIS
LIN {X 0.080,Y -418.033,Z 1043.859,A 0.000,B 0.000,C 90.000,E1 190.602} C_DIS
LIN {X 0.138,Y -419.435,Z 1043.857,A 0.000,B 0.000,C 90.000,E1 190.254} C_DIS
LIN {X 0.227,Y -424.691,Z 1043.852,A 0.000,B 0.000,C 90.000,E1 189.321} C_DIS
LIN {X -0.197,Y -439.313,Z 1043.840,A 0.000,B 0.000,C 90.000,E1 187.239} C_DIS
LIN {X -0.175,Y -447.663,Z 1043.834,A 0.000,B 0.000,C 90.000,E1 186.087} C_DIS
LIN {X 0.092,Y -457.232,Z 1043.827,A 0.000,B 0.000,C 90.000,E1 184.759} C_DIS
LIN {X 0.130,Y -462.954,Z 1043.822,A 0.000,B 0.000,C 90.000,E1 183.955} C_DIS
LIN {X -0.018,Y -470.516,Z 1043.816,A 0.000,B 0.000,C 90.000,E1 182.865} C_DIS
LIN {X 0.130,Y -475.760,Z 1043.812,A 0.000,B 0.000,C 90.000,E1 182.064} C_DIS
LIN {X -0.226,Y -481.673,Z 1043.807,A 0.000,B 0.000,C 90.000,E1 181.203} C_DIS
LIN {X 0.189,Y -487.556,Z 1043.801,A 0.000,B 0.000,C 90.000,E1 180.229} C_DIS
LIN {X -0.102,Y -494.182,Z 1043.796,A 0.000,B 0.000,C 90.000,E1 179.198} C_DIS
LIN {X -0.032,Y -499.807,Z 1043.791,A 0.000,B 0.000,C 90.000,E1 178.282} C_DIS
LIN {X -0.254,Y -507.629,Z 1043.783,A 0.000,B 0.000,C 90.000,E1 176.963} C_DIS
LIN {X -0.149,Y -516.149,Z 1043.775,A 0.000,B 0.000,C 90.000,E1 175.469} C_DIS
LIN {X 0.178,Y -522.855,Z 1043.768,A 0.000,B 0.000,C 90.000,E1 174.261} C_DIS
LIN {X 0.107,Y -531.093,Z 1043.760,A 0.000,B 0.000,C 90.000,E1 172.818} C_DIS
LIN {X -0.075,Y -538.224,Z 1043.753,A 0.000,B 0.000,C 90.000,E1 171.546} C_DIS
LIN {X -0.150,Y -545.273,Z 1043.746,A 0.000,B 0.000,C 90.000,E1 170.274} C_DIS
LIN {X -0.186,Y -553.003,Z 1043.738,A 0.000,B 0.000,C 90.000,E1 168.870} C_DIS
LIN {X 0.064,Y -559.673,Z 1043.731,A 0.000,B 0.000,C 90.000,E1 167.589} C_DIS
LIN {X -0.008,Y -566.191,Z 1043.724,A 0.000,B 0.000,C 90.000,E1 166.353} C_DIS
LIN {X -0.163,Y -571.009,Z 1043.719,A 0.000,B 0.000,C 90.000,E1 165.408} C_DIS
LIN {X 0.189,Y -576.329,Z 1043.713,A 0.000,B 0.000,C 90.000,E1 164.283} C_DIS
LIN {X 0.226,Y -581.544,Z 1043.707,A 0.000,B 0.000,C 90.000,E1 163.196} C_DIS
LIN {X 0.165,Y -586.342,Z 1043.701,A 0.000,B 0.000,C 90.000,E1 162.127} C_DIS
LIN {X -0.217,Y -590.833,Z 1043.695,A 0.000,B 0.000,C 90.000,E1 161.094} C_DIS
LIN {X 0.333,Y -594.042,Z 1043.690,A 0.000,B 0.000,C 90.000,E1 160.242} C_DIS
LIN {X 0.154,Y -597.132,Z 1043.686,A 0.000,B 0.000,C 90.000,E1 159.464} C_DIS
LIN {X -0.349,Y -600.052,Z 1043.682,A 0.000,B 0.000,C 90.000,E1 158.720} C_DIS
LIN {X 0.220,Y -603.703,Z 1043.676,A 0.000,B 0.000,C 90.000,E1 157.614} C_DIS
LIN {X -0.277,Y -607.133,Z 1043.670,A 0.000,B 0.000,C 90.000,E1 156.613} C_DIS
LIN {X 0.078,Y -610.351,Z 1043.664,A 0.000,B 0.000,C 90.000,E1 155.537} C_DIS
LIN {X -0.298,Y -612.687,Z 1043.660,A 0.000,B 0.000,C 90.000,E1 154.793} C_DIS
LIN {X 0.110,Y -616.230,Z 1043.653,A 0.000,B 0.000,C 90.000,E1 153.461} C_DIS
LIN {X 0.300,Y -620.257,Z 1043.644,A 0.000,B 0.000,C 90.000,E1 151.897} C_DIS
LIN {X -0.270,Y -623.383,Z 1043.637,A 0.000,B 0.000,C 90.000,E1 150.667} C_DIS
LIN {X 0.046,Y -625.961,Z 1043.631,A 0.000,B 0.000,C 90.000,E1 149.616} C_DIS
LIN {X 0.203,Y -629.562,Z 1043.623,A 0.000,B 0.000,C 90.000,E1 148.074} C_DIS
LIN {X 0.399,Y -631.875,Z 1043.617,A 0.000,B 0.000,C 90.000,E1 147.041} C_DIS
LIN {X 0.123,Y -634.761,Z 1043.610,A 0.000,B 0.000,C 90.000,E1 145.801} C_DIS
LIN {X 0.275,Y -638.147,Z 1043.602,A 0.000,B 0.000,C 90.000,E1 144.276} C_DIS
LIN {X 0.061,Y -640.414,Z 1043.596,A 0.000,B 0.000,C 90.000,E1 143.290} C_DIS
LIN {X -0.329,Y -643.800,Z 1043.588,A 0.000,B 0.000,C 90.000,E1 141.823} C_DIS
LIN {X -0.228,Y -647.767,Z 1043.578,A 0.000,B 0.000,C 90.000,E1 140.070} C_DIS
LIN {X -0.005,Y -649.955,Z 1043.573,A 0.000,B 0.000,C 90.000,E1 139.057} C_DIS
LIN {X 0.209,Y -653.282,Z 1043.564,A 0.000,B 0.000,C 90.000,E1 137.553} C_DIS
LIN {X 0.379,Y -658.060,Z 1043.553,A 0.000,B 0.000,C 90.000,E1 135.567} C_DIS
LIN {X 0.182,Y -664.693,Z 1043.540,A 0.000,B 0.000,C 90.000,E1 133.137} C_DIS
LIN {X -0.246,Y -670.771,Z 1043.528,A 0.000,B 0.000,C 90.000,E1 130.987} C_DIS
LIN {X -0.014,Y -676.097,Z 1043.517,A 0.000,B 0.000,C 90.000,E1 129.036} C_DIS
LIN {X 0.132,Y -678.078,Z 1043.513,A 0.000,B 0.000,C 90.000,E1 128.302} C_DIS
LIN {X 0.067,Y -681.727,Z 1043.505,A 0.000,B 0.000,C 90.000,E1 126.870} C_DIS
LIN {X -0.307,Y -685.982,Z 1043.496,A 0.000,B 0.000,C 90.000,E1 125.231} C_DIS
LIN {X -0.419,Y -690.261,Z 1043.486,A 0.000,B 0.000,C 90.000,E1 123.579} C_DIS
LIN {X 0.272,Y -693.081,Z 1043.480,A 0.000,B 0.000,C 90.000,E1 122.339} C_DIS
LIN {X 0.043,Y -695.841,Z 1043.473,A 0.000,B 0.000,C 90.000,E1 121.180} C_DIS
LIN {X 0.188,Y -697.345,Z 1043.469,A 0.000,B 0.000,C 90.000,E1 120.463} C_DIS
LIN {X 0.009,Y -698.989,Z 1043.464,A 0.000,B 0.000,C 90.000,E1 119.539} C_DIS
LIN {X 0.192,Y -700.000,Z 1043.460,A 0.000,B 0.000,C 90.000,E1 118.821} C_DIS
LIN {X -0.034,Y -701.617,Z 1043.453,A 0.000,B 0.000,C 90.000,E1 117.436} C_DIS
LIN {X -0.220,Y -702.918,Z 1043.446,A 0.000,B 0.000,C 90.000,E1 116.283} C_DIS
LIN {X -0.035,Y -703.752,Z 1043.441,A 0.000,B 0.000,C 90.000,E1 115.335} C_DIS
LIN {X -0.122,Y -704.145,Z 1043.437,A 0.000,B 0.000,C 90.000,E1 114.643} C_DIS
LIN {X 0.156,Y -703.991,Z 1043.434,A 0.000,B 0.000,C 90.000,E1 114.155} C_DIS
LIN {X -0.204,Y -703.646,Z 1043.433,A 0.000,B 0.000,C 90.000,E1 113.951} C_DIS
LIN {X 0.076,Y -702.556,Z 1043.430,A 0.000,B 0.000,C 90.000,E1 113.462} C_DIS
LIN {X -0.291,Y -701.382,Z 1043.429,A 0.000,B 0.000,C 90.000,E1 113.259} C_DIS
LIN {X -0.024,Y -698.402,Z 1043.427,A 0.000,B 0.000,C 90.000,E1 112.770} C_DIS
LIN {X 0.106,Y -697.206,Z 1043.426,A 0.000,B 0.000,C 90.000,E1 112.642} C_DIS
LIN {X 0.236,Y -695.366,Z 1043.425,A 0.000,B 0.000,C 90.000,E1 112.514} C_DIS
LIN {X -0.196,Y -688.571,Z 1043.423,A 0.000,B 0.000,C 90.000,E1 112.206} C_DIS
LIN {X 0.131,Y -686.317,Z 1043.423,A 0.000,B 0.000,C 90.000,E1 112.099} C_DIS
LIN {X 0.079,Y -682.927,Z 1043.422,A 0.000,B 0.000,C 90.000,E1 112.025} C_DIS
LIN {X -0.083,Y -675.848,Z 1043.422,A 0.000,B 0.000,C 90.000,E1 111.950} C_DIS
LIN {X -0.135,Y -610.889,Z 1043.422,A 0.000,B 0.000,C 90.000,E1 111.950} C_DIS
LIN {X 0.079,Y -604.650,Z 1043.421,A 0.000,B 0.000,C 90.000,E1 111.716} C_DIS
LIN {X -0.012,Y -598.303,Z 1043.419,A 0.000,B 0.000,C 90.000,E1 111.408} C_DIS
LIN {X 0.128,Y -595.614,Z 1043.418,A 0.000,B 0.000,C 90.000,E1 111.227} C_DIS
LIN {X 0.168,Y -591.272,Z 1043.416,A 0.000,B 0.000,C 90.000,E1 110.918} C_DIS
LIN {X 0.062,Y -576.250,Z 1043.410,A 0.000,B 0.000,C 90.000,E1 109.704} C_DIS
LIN {X -0.140,Y -570.141,Z 1043.407,A 0.000,B 0.000,C 90.000,E1 109.268} C_DIS
LIN {X 0.021,Y -563.425,Z 1043.405,A 0.000,B 0.000,C 90.000,E1 108.852} C_DIS
LIN {X 0.088,Y -553.805,Z 1043.402,A 0.000,B 0.000,C 90.000,E1 108.308} C_DIS
LIN {X 0.255,Y -549.435,Z 1043.400,A 0.000,B 0.000,C 90.000,E1 108.000} C_DIS
LIN {X 0.234,Y -547.935,Z 1043.399,A 0.000,B 0.000,C 90.000,E1 107.819} C_DIS
LIN {X 0.193,Y -547.907,Z 1043.399,A 0.000,B 0.000,C 90.000,E1 107.819} C_DIS
LIN {X -0.241,Y -547.483,Z 1043.398,A 0.000,B 0.000,C 90.000,E1 107.583} C_DIS
LIN {X -0.106,Y -547.589,Z 1043.394,A 0.000,B 0.000,C 90.000,E1 106.968} C_DIS
LIN {X -0.115,Y -548.252,Z 1043.388,A 0.000,B 0.000,C 90.000,E1 105.843} C_DIS
LIN {X 0.233,Y -549.246,Z 1043.379,A 0.000,B 0.000,C 90.000,E1 104.120} C_DIS
LIN {X -0.162,Y -551.668,Z 1043.361,A 0.000,B 0.000,C 90.000,E1 101.074} C_DIS
LIN {X 0.157,Y -554.040,Z 1043.349,A 0.000,B 0.000,C 90.000,E1 98.803} C_DIS
LIN {X -0.232,Y -556.278,Z 1043.338,A 0.000,B 0.000,C 90.000,E1 96.891} C_DIS
LIN {X 0.142,Y -557.526,Z 1043.332,A 0.000,B 0.000,C 90.000,E1 95.739} C_DIS
LIN {X 0.055,Y -558.702,Z 1043.324,A 0.000,B 0.000,C 90.000,E1 94.359} C_DIS
LIN {X -0.133,Y -559.486,Z 1043.318,A 0.000,B 0.000,C 90.000,E1 93.269} C_DIS
LIN {X -0.217,Y -560.223,Z 1043.310,A 0.000,B 0.000,C 90.000,E1 91.892} C_DIS
LIN {X 0.078,Y -560.556,Z 1043.306,A 0.000,B 0.000,C 90.000,E1 91.031} C_DIS
LIN {X 0.090,Y -561.139,Z 1043.297,A 0.000,B 0.000,C 90.000,E1 89.370} C_DIS
LIN {X 0.223,Y -561.738,Z 1043.286,A 0.000,B 0.000,C 90.000,E1 87.421} C_DIS
LIN {X -0.258,Y -562.354,Z 1043.277,A 0.000,B 0.000,C 90.000,E1 85.812} C_DIS
LIN {X -0.259,Y -562.768,Z 1043.269,A 0.000,B 0.000,C 90.000,E1 84.432} C_DIS
LIN {X 0.044,Y -563.228,Z 1043.258,A 0.000,B 0.000,C 90.000,E1 82.470} C_DIS
LIN {X 0.105,Y -563.991,Z 1043.245,A 0.000,B 0.000,C 90.000,E1 79.982} C_DIS
LIN {X -0.067,Y -565.073,Z 1043.231,A 0.000,B 0.000,C 90.000,E1 77.521} C_DIS
LIN {X 0.003,Y -566.182,Z 1043.220,A 0.000,B 0.000,C 90.000,E1 75.589} C_DIS
LIN {X -0.233,Y -567.928,Z 1043.206,A 0.000,B 0.000,C 90.000,E1 73.142} C_DIS
LIN {X -0.163,Y -569.042,Z 1043.199,A 0.000,B 0.000,C 90.000,E1 71.764} C_DIS
LIN {X -0.084,Y -570.434,Z 1043.190,A 0.000,B 0.000,C 90.000,E1 70.115} C_DIS
LIN {X 0.208,Y -571.389,Z 1043.182,A 0.000,B 0.000,C 90.000,E1 68.720} C_DIS
LIN {X 0.185,Y -572.384,Z 1043.174,A 0.000,B 0.000,C 90.000,E1 67.358} C_DIS
LIN {X 0.010,Y -573.409,Z 1043.165,A 0.000,B 0.000,C 90.000,E1 65.741} C_DIS
LIN {X 0.084,Y -574.292,Z 1043.156,A 0.000,B 0.000,C 90.000,E1 64.101} C_DIS
LIN {X -0.240,Y -575.235,Z 1043.146,A 0.000,B 0.000,C 90.000,E1 62.231} C_DIS
LIN {X -0.268,Y -576.023,Z 1043.135,A 0.000,B 0.000,C 90.000,E1 60.333} C_DIS
LIN {X 0.167,Y -576.764,Z 1043.126,A 0.000,B 0.000,C 90.000,E1 58.663} C_DIS
LIN {X -0.022,Y -577.261,Z 1043.119,A 0.000,B 0.000,C 90.000,E1 57.327} C_DIS
LIN {X 0.255,Y -577.666,Z 1043.109,A 0.000,B 0.000,C 90.000,E1 55.674} C_DIS
LIN {X 0.064,Y -577.930,Z 1043.100,A 0.000,B 0.000,C 90.000,E1 54.069} C_DIS
LIN {X -0.108,Y -577.992,Z 1043.094,A 0.000,B 0.000,C 90.000,E1 53.004} C_DIS
LIN {X -0.088,Y -577.908,Z 1043.090,A 0.000,B 0.000,C 90.000,E1 52.190} C_DIS
LIN {X -0.063,Y -577.712,Z 1043.085,A 0.000,B 0.000,C 90.000,E1 51.376} C_DIS
LIN {X -0.015,Y -577.007,Z 1043.076,A 0.000,B 0.000,C 90.000,E1 49.747} C_DIS
LIN {X 0.001,Y -576.115,Z 1043.067,A 0.000,B 0.000,C 90.000,E1 48.119} C_DIS
LIN {X 0.091,Y -575.282,Z 1043.061,A 0.000,B 0.000,C 90.000,E1 47.025} C_DIS
LIN {X 0.043,Y -574.550,Z 1043.057,A 0.000,B 0.000,C 90.000,E1 46.215} C_DIS
LIN {X -0.008,Y -573.631,Z 1043.052,A 0.000,B 0.000,C 90.000,E1 45.405} C_DIS
LIN {X -0.067,Y -572.533,Z 1043.048,A 0.000,B 0.000,C 90.000,E1 44.595} C_DIS
LIN {X -0.139,Y -571.279,Z 1043.043,A 0.000,B 0.000,C 90.000,E1 43.785} C_DIS
LIN {X -0.113,Y -569.443,Z 1043.037,A 0.000,B 0.000,C 90.000,E1 42.690} C_DIS
LIN {X 0.196,Y -567.875,Z 1043.033,A 0.000,B 0.000,C 90.000,E1 41.838} C_DIS
LIN {X -0.203,Y -565.407,Z 1043.026,A 0.000,B 0.000,C 90.000,E1 40.782} C_DIS
LIN {X -0.049,Y -564.086,Z 1043.023,A 0.000,B 0.000,C 90.000,E1 40.216} C_DIS
LIN {X -0.072,Y -561.069,Z 1043.017,A 0.000,B 0.000,C 90.000,E1 39.116} C_DIS
LIN {X 0.214,Y -558.397,Z 1043.013,A 0.000,B 0.000,C 90.000,E1 38.257} C_DIS
LIN {X 0.113,Y -554.429,Z 1043.007,A 0.000,B 0.000,C 90.000,E1 37.156} C_DIS
LIN {X 0.328,Y -551.022,Z 1043.002,A 0.000,B 0.000,C 90.000,E1 36.297} C_DIS
LIN {X -0.131,Y -547.886,Z 1042.998,A 0.000,B 0.000,C 90.000,E1 35.644} C_DIS
LIN {X 0.308,Y -543.207,Z 1042.993,A 0.000,B 0.000,C 90.000,E1 34.612} C_DIS
LIN {X 0.221,Y -539.588,Z 1042.989,A 0.000,B 0.000,C 90.000,E1 33.913} C_DIS
LIN {X -0.192,Y -534.232,Z 1042.983,A 0.000,B 0.000,C 90.000,E1 32.959} C_DIS
LIN {X 0.087,Y -529.982,Z 1042.979,A 0.000,B 0.000,C 90.000,E1 32.212} C_DIS
LIN {X -0.123,Y -525.562,Z 1042.975,A 0.000,B 0.000,C 90.000,E1 31.514} C_DIS
LIN {X 0.121,Y -522.728,Z 1042.973,A 0.000,B 0.000,C 90.000,E1 31.052} C_DIS
LIN {X 0.185,Y -518.770,Z 1042.969,A 0.000,B 0.000,C 90.000,E1 30.463} C_DIS
LIN {X 0.221,Y -514.578,Z 1042.966,A 0.000,B 0.000,C 90.000,E1 29.873} C_DIS
LIN {X -0.040,Y -511.286,Z 1042.964,A 0.000,B 0.000,C 90.000,E1 29.461} C_DIS
LIN {X -0.058,Y -506.526,Z 1042.960,A 0.000,B 0.000,C 90.000,E1 28.871} C_DIS
LIN {X 0.083,Y -501.712,Z 1042.957,A 0.000,B 0.000,C 90.000,E1 28.281} C_DIS
LIN {X -0.008,Y -495.018,Z 1042.953,A 0.000,B 0.000,C 90.000,E1 27.564} C_DIS
LIN {X 0.090,Y -486.763,Z 1042.948,A 0.000,B 0.000,C 90.000,E1 26.693} C_DIS
LIN {X -0.046,Y -475.285,Z 1042.942,A 0.000,B 0.000,C 90.000,E1 25.591} C_DIS
LIN {X -0.039,Y -464.967,Z 1042.937,A 0.000,B 0.000,C 90.000,E1 24.643} C_DIS
LIN {X 0.054,Y -454.361,Z 1042.932,A 0.000,B 0.000,C 90.000,E1 23.718} C_DIS
LIN {X -0.053,Y -430.494,Z 1042.920,A 0.000,B 0.000,C 90.000,E1 21.642} C_DIS
LIN {X 0.070,Y -418.781,Z 1042.914,A 0.000,B 0.000,C 90.000,E1 20.482} C_DIS
LIN {X 0.185,Y -406.155,Z 1042.906,A 0.000,B 0.000,C 90.000,E1 19.087} C_DIS
LIN {X -0.113,Y -400.764,Z 1042.903,A 0.000,B 0.000,C 90.000,E1 18.471} C_DIS
LIN {X -0.105,Y -396.845,Z 1042.900,A 0.000,B 0.000,C 90.000,E1 17.946} C_DIS
LIN {X 0.048,Y -394.141,Z 1042.897,A 0.000,B 0.000,C 90.000,E1 17.457} C_DIS
LIN {X 0.169,Y -392.172,Z 1042.894,A 0.000,B 0.000,C 90.000,E1 16.913} C_DIS
LIN {X 0.133,Y -391.383,Z 1042.891,A 0.000,B 0.000,C 90.000,E1 16.386} C_DIS
LIN {X 0.201,Y -391.355,Z 1042.888,A 0.000,B 0.000,C 90.000,E1 15.843} C_DIS
LIN {X -0.150,Y -392.202,Z 1042.882,A 0.000,B 0.000,C 90.000,E1 14.828} C_DIS
LIN {X 0.050,Y -398.759,Z 1042.855,A 0.000,B 0.000,C 90.000,E1 9.849} C_DIS
LIN {X -0.108,Y -405.154,Z 1042.835,A 0.000,B 0.000,C 90.000,E1 6.372} C_DIS
LIN {X -0.166,Y -408.891,Z 1042.826,A 0.000,B 0.000,C 90.000,E1 4.645} C_DIS
LIN {X -0.201,Y -412.009,Z 1042.818,A 0.000,B 0.000,C 90.000,E1 3.269} C_DIS
LIN {X -0.185,Y -413.946,Z 1042.815,A 0.000,B 0.000,C 90.000,E1 2.751} C_DIS
LIN {X -0.185,Y -414.836,Z 1042.814,A 0.000,B 0.000,C 90.000,E1 2.579} C_DIS
LIN {X -0.163,Y -418.194,Z 1042.811,A 0.000,B 0.000,C 90.000,E1 2.064} C_DIS
LIN {X 0.016,Y -421.386,Z 1042.810,A 0.000,B 0.000,C 90.000,E1 1.718} C_DIS
LIN {X 0.186,Y -423.185,Z 1042.809,A 0.000,B 0.000,C 90.000,E1 1.547} C_DIS
LIN {X 0.040,Y -438.702,Z 1042.803,A 0.000,B 0.000,C 90.000,E1 0.573} C_DIS
LIN {X -0.086,Y -454.572,Z 1042.798,A 0.000,B 0.000,C 90.000,E1 359.599} C_DIS
LIN {X 0.218,Y -472.797,Z 1042.792,A 0.000,B 0.000,C 90.000,E1 358.453} C_DIS
LIN {X -0.186,Y -485.939,Z 1042.787,A 0.000,B 0.000,C 90.000,E1 357.707} C_DIS
LIN {X 0.238,Y -497.249,Z 1042.783,A 0.000,B 0.000,C 90.000,E1 356.963} C_DIS
LIN {X 0.223,Y -505.077,Z 1042.780,A 0.000,B 0.000,C 90.000,E1 356.445} C_DIS
LIN {X 0.089,Y -515.877,Z 1042.776,A 0.000,B 0.000,C 90.000,E1 355.698} C_DIS
LIN {X 0.084,Y -524.619,Z 1042.772,A 0.000,B 0.000,C 90.000,E1 355.008} C_DIS
LIN {X -0.240,Y -531.740,Z 1042.769,A 0.000,B 0.000,C 90.000,E1 354.432} C_DIS
LIN {X 0.164,Y -538.519,Z 1042.765,A 0.000,B 0.000,C 90.000,E1 353.742} C_DIS
LIN {X -0.210,Y -544.872,Z 1042.762,A 0.000,B 0.000,C 90.000,E1 353.109} C_DIS
LIN {X -0.049,Y -549.772,Z 1042.759,A 0.000,B 0.000,C 90.000,E1 352.534} C_DIS
LIN {X -0.095,Y -555.280,Z 1042.755,A 0.000,B 0.000,C 90.000,E1 351.837} C_DIS
LIN {X 0.162,Y -559.218,Z 1042.752,A 0.000,B 0.000,C 90.000,E1 351.254} C_DIS
LIN {X 0.116,Y -563.640,Z 1042.748,A 0.000,B 0.000,C 90.000,E1 350.566} C_DIS
LIN {X 0.053,Y -568.443,Z 1042.743,A 0.000,B 0.000,C 90.000,E1 349.746} C_DIS
LIN {X 0.046,Y -572.924,Z 1042.739,A 0.000,B 0.000,C 90.000,E1 348.926} C_DIS
LIN {X -0.029,Y -576.965,Z 1042.734,A 0.000,B 0.000,C 90.000,E1 348.117} C_DIS
LIN {X 0.286,Y -580.065,Z 1042.730,A 0.000,B 0.000,C 90.000,E1 347.409} C_DIS
LIN {X 0.062,Y -584.710,Z 1042.724,A 0.000,B 0.000,C 90.000,E1 346.353} C_DIS
LIN {X -0.210,Y -587.962,Z 1042.720,A 0.000,B 0.000,C 90.000,E1 345.574} C_DIS
LIN {X 0.082,Y -593.254,Z 1042.712,A 0.000,B 0.000,C 90.000,E1 344.212} C_DIS
LIN {X 0.183,Y -597.281,Z 1042.707,A 0.000,B 0.000,C 90.000,E1 343.142} C_DIS
LIN {X 0.048,Y -600.144,Z 1042.702,A 0.000,B 0.000,C 90.000,E1 342.362} C_DIS
LIN {X 0.138,Y -604.609,Z 1042.695,A 0.000,B 0.000,C 90.000,E1 341.040} C_DIS
LIN {X -0.005,Y -607.813,Z 1042.689,A 0.000,B 0.000,C 90.000,E1 340.007} C_DIS
LIN {X 0.111,Y -610.839,Z 1042.683,A 0.000,B 0.000,C 90.000,E1 338.954} C_DIS
LIN {X 0.047,Y -613.578,Z 1042.677,A 0.000,B 0.000,C 90.000,E1 337.922} C_DIS
LIN {X -0.323,Y -616.174,Z 1042.672,A 0.000,B 0.000,C 90.000,E1 336.922} C_DIS
LIN {X -0.110,Y -619.125,Z 1042.665,A 0.000,B 0.000,C 90.000,E1 335.613} C_DIS
LIN {X -0.150,Y -621.618,Z 1042.657,A 0.000,B 0.000,C 90.000,E1 334.332} C_DIS
LIN {X -0.147,Y -623.019,Z 1042.653,A 0.000,B 0.000,C 90.000,E1 333.563} C_DIS
LIN {X -0.114,Y -625.073,Z 1042.646,A 0.000,B 0.000,C 90.000,E1 332.281} C_DIS
LIN {X -0.071,Y -626.539,Z 1042.640,A 0.000,B 0.000,C 90.000,E1 331.257} C_DIS
LIN {X -0.242,Y -628.126,Z 1042.633,A 0.000,B 0.000,C 90.000,E1 329.999} C_DIS
LIN {X -0.387,Y -629.347,Z 1042.626,A 0.000,B 0.000,C 90.000,E1 328.742} C_DIS
LIN {X -0.186,Y -630.352,Z 1042.619,A 0.000,B 0.000,C 90.000,E1 327.454} C_DIS
LIN {X 0.026,Y -631.009,Z 1042.612,A 0.000,B 0.000,C 90.000,E1 326.167} C_DIS
LIN {X 0.080,Y -631.271,Z 1042.605,A 0.000,B 0.000,C 90.000,E1 324.895} C_DIS
LIN {X -0.372,Y -631.359,Z 1042.597,A 0.000,B 0.000,C 90.000,E1 323.417} C_DIS
LIN {X -0.085,Y -631.449,Z 1042.587,A 0.000,B 0.000,C 90.000,E1 321.618} C_DIS
LIN {X -0.134,Y -631.597,Z 1042.580,A 0.000,B 0.000,C 90.000,E1 320.356} C_DIS
LIN {X -0.182,Y -631.801,Z 1042.573,A 0.000,B 0.000,C 90.000,E1 319.094} C_DIS
LIN {X 0.181,Y -631.845,Z 1042.566,A 0.000,B 0.000,C 90.000,E1 317.796} C_DIS
LIN {X -0.256,Y -632.050,Z 1042.554,A 0.000,B 0.000,C 90.000,E1 315.810} C_DIS
LIN {X -0.020,Y -632.267,Z 1042.546,A 0.000,B 0.000,C 90.000,E1 314.271} C_DIS
LIN {X -0.332,Y -632.530,Z 1042.536,A 0.000,B 0.000,C 90.000,E1 312.528} C_DIS
LIN {X -0.067,Y -632.601,Z 1042.528,A 0.000,B 0.000,C 90.000,E1 310.987} C_DIS
LIN {X -0.097,Y -632.647,Z 1042.521,A 0.000,B 0.000,C 90.000,E1 309.725} C_DIS
LIN {X -0.001,Y -632.620,Z 1042.515,A 0.000,B 0.000,C 90.000,E1 308.705} C_DIS
LIN {X -0.176,Y -632.556,Z 1042.505,A 0.000,B 0.000,C 90.000,E1 306.950} C_DIS
LIN {X 0.057,Y -632.586,Z 1042.502,A 0.000,B 0.000,C 90.000,E1 306.423} C_DIS
LIN {X -0.233,Y -632.696,Z 1042.497,A 0.000,B 0.000,C 90.000,E1 305.438} C_DIS
LIN {X 0.122,Y -633.630,Z 1042.481,A 0.000,B 0.000,C 90.000,E1 302.625} C_DIS
LIN {X 0.283,Y -634.612,Z 1042.470,A 0.000,B 0.000,C 90.000,E1 300.590} C_DIS
LIN {X 0.287,Y -635.704,Z 1042.462,A 0.000,B 0.000,C 90.000,E1 299.077} C_DIS
LIN {X 0.012,Y -636.824,Z 1042.453,A 0.000,B 0.000,C 90.000,E1 297.590} C_DIS
LIN {X -0.348,Y -637.514,Z 1042.448,A 0.000,B 0.000,C 90.000,E1 296.616} C_DIS
LIN {X -0.188,Y -637.822,Z 1042.444,A 0.000,B 0.000,C 90.000,E1 295.848} C_DIS
LIN {X -0.080,Y -637.972,Z 1042.441,A 0.000,B 0.000,C 90.000,E1 295.335} C_DIS
LIN {X -0.081,Y -637.934,Z 1042.434,A 0.000,B 0.000,C 90.000,E1 294.079} C_DIS
LIN {X -0.182,Y -637.575,Z 1042.430,A 0.000,B 0.000,C 90.000,E1 293.334} C_DIS
LIN {X -0.238,Y -637.171,Z 1042.424,A 0.000,B 0.000,C 90.000,E1 292.333} C_DIS
LIN {X -0.389,Y -636.615,Z 1042.421,A 0.000,B 0.000,C 90.000,E1 291.844} C_DIS
LIN {X 0.283,Y -635.805,Z 1042.418,A 0.000,B 0.000,C 90.000,E1 291.280} C_DIS
LIN {X 0.090,Y -635.261,Z 1042.417,A 0.000,B 0.000,C 90.000,E1 291.046} C_DIS
LIN {X -0.068,Y -633.618,Z 1042.414,A 0.000,B 0.000,C 90.000,E1 290.556} C_DIS
LIN {X -0.041,Y -632.286,Z 1042.413,A 0.000,B 0.000,C 90.000,E1 290.301} C_DIS
LIN {X -0.230,Y -629.874,Z 1042.411,A 0.000,B 0.000,C 90.000,E1 289.939} C_DIS
LIN {X -0.219,Y -627.538,Z 1042.409,A 0.000,B 0.000,C 90.000,E1 289.685} C_DIS
LIN {X 0.266,Y -623.545,Z 1042.407,A 0.000,B 0.000,C 90.000,E1 289.268} C_DIS
LIN {X 0.170,Y -616.692,Z 1042.405,A 0.000,B 0.000,C 90.000,E1 288.852} C_DIS
LIN {X -0.064,Y -614.983,Z 1042.404,A 0.000,B 0.000,C 90.000,E1 288.779} C_DIS
LIN {X -0.112,Y -605.741,Z 1042.402,A 0.000,B 0.000,C 90.000,E1 288.417} C_DIS
LIN {X 0.229,Y -595.066,Z 1042.400,A 0.000,B 0.000,C 90.000,E1 288.000} C_DIS
LIN {X 0.248,Y -589.528,Z 1042.399,A 0.000,B 0.000,C 90.000,E1 287.819} C_DIS
LIN {X 0.128,Y -573.799,Z 1042.396,A 0.000,B 0.000,C 90.000,E1 287.347} C_DIS
LIN {X -0.312,Y -563.915,Z 1042.395,A 0.000,B 0.000,C 90.000,E1 287.040} C_DIS
LIN {X 0.215,Y -558.157,Z 1042.393,A 0.000,B 0.000,C 90.000,E1 286.732} C_DIS
LIN {X -0.155,Y -554.167,Z 1042.392,A 0.000,B 0.000,C 90.000,E1 286.551} C_DIS
LIN {X 0.093,Y -552.627,Z 1042.391,A 0.000,B 0.000,C 90.000,E1 286.315} C_DIS
LIN {X -0.129,Y -551.858,Z 1042.390,A 0.000,B 0.000,C 90.000,E1 286.205} C_DIS
LIN {X -0.188,Y -550.420,Z 1042.388,A 0.000,B 0.000,C 90.000,E1 285.788} C_DIS
LIN {X 0.171,Y -549.431,Z 1042.385,A 0.000,B 0.000,C 90.000,E1 285.190} C_DIS
LIN {X -0.211,Y -549.003,Z 1042.382,A 0.000,B 0.000,C 90.000,E1 284.828} C_DIS
LIN {X 0.296,Y -588.864,Z 1042.382,A 0.000,B 0.000,C 90.000,E1 284.773} C_DIS
LIN {X 0.127,Y -589.495,Z 1042.382,A 0.000,B 0.000,C 90.000,E1 284.773} C_DIS
LIN {X -0.013,Y -591.791,Z 1042.381,A 0.000,B 0.000,C 90.000,E1 284.647} C_DIS
LIN {X -0.255,Y -594.373,Z 1042.380,A 0.000,B 0.000,C 90.000,E1 284.481} C_DIS
LIN {X -0.027,Y -596.553,Z 1042.379,A 0.000,B 0.000,C 90.000,E1 284.245} C_DIS
LIN {X -0.045,Y -597.505,Z 1042.378,A 0.000,B 0.000,C 90.000,E1 284.120} C_DIS
LIN {X 0.084,Y -599.640,Z 1042.376,A 0.000,B 0.000,C 90.000,E1 283.716} C_DIS
LIN {X 0.012,Y -600.332,Z 1042.376,A 0.000,B 0.000,C 90.000,E1 283.592} C_DIS
LIN {X -0.061,Y -600.873,Z 1042.375,A 0.000,B 0.000,C 90.000,E1 283.467} C_DIS
LIN {X 0.242,Y -601.574,Z 1042.373,A 0.000,B 0.000,C 90.000,E1 283.175} C_DIS
LIN {X 0.268,Y -602.469,Z 1042.370,A 0.000,B 0.000,C 90.000,E1 282.647} C_DIS
LIN {X 0.303,Y -602.728,Z 1042.368,A 0.000,B 0.000,C 90.000,E1 282.119} C_DIS
LIN {X 0.026,Y -602.511,Z 1042.366,A 0.000,B 0.000,C 90.000,E1 281.883} C_DIS
LIN {X 0.218,Y -602.126,Z 1042.365,A 0.000,B 0.000,C 90.000,E1 281.602} C_DIS
LIN {X -0.058,Y -601.535,Z 1042.363,A 0.000,B 0.000,C 90.000,E1 281.366} C_DIS
LIN {X -0.026,Y -599.520,Z 1042.360,A 0.000,B 0.000,C 90.000,E1 280.838} C_DIS
LIN {X -0.011,Y -596.440,Z 1042.357,A 0.000,B 0.000,C 90.000,E1 280.310} C_DIS
LIN {X -0.124,Y -592.629,Z 1042.354,A 0.000,B 0.000,C 90.000,E1 279.792} C_DIS
LIN {X -0.227,Y -591.235,Z 1042.354,A 0.000,B 0.000,C 90.000,E1 279.670} C_DIS
LIN {X 0.153,Y -589.632,Z 1042.353,A 0.000,B 0.000,C 90.000,E1 279.500} C_DIS
LIN {X 0.157,Y -586.240,Z 1042.351,A 0.000,B 0.000,C 90.000,E1 279.151} C_DIS
LIN {X 0.204,Y -584.679,Z 1042.350,A 0.000,B 0.000,C 90.000,E1 279.029} C_DIS
LIN {X 0.015,Y -576.820,Z 1042.348,A 0.000,B 0.000,C 90.000,E1 278.681} C_DIS
LIN {X -0.251,Y -570.290,Z 1042.348,A 0.000,B 0.000,C 90.000,E1 278.624} C_DIS
LIN {X 0.266,Y -544.283,Z 1042.348,A 0.000,B 0.000,C 90.000,E1 278.568} C_DIS
LIN {X -0.145,Y -543.695,Z 1042.344,A 0.000,B 0.000,C 90.000,E1 277.936} C_DIS
LIN {X -0.187,Y -543.692,Z 1042.344,A 0.000,B 0.000,C 90.000,E1 277.936} C_DIS
LIN {X -0.223,Y -544.175,Z 1042.343,A 0.000,B 0.000,C 90.000,E1 277.701} C_DIS
LIN {X -0.142,Y -543.823,Z 1042.341,A 0.000,B 0.000,C 90.000,E1 277.409} C_DIS
LIN {X -0.118,Y -543.007,Z 1042.340,A 0.000,B 0.000,C 90.000,E1 277.239} C_DIS
LIN {X -0.159,Y -543.001,Z 1042.340,A 0.000,B 0.000,C 90.000,E1 277.239} C_DIS
LIN {X 0.196,Y -541.383,Z 1042.328,A 0.000,B 0.000,C 90.000,E1 275.106} C_DIS
LIN {X -0.181,Y -540.500,Z 1042.321,A 0.000,B 0.000,C 90.000,E1 273.726} C_DIS
LIN {X -0.015,Y -539.371,Z 1042.310,A 0.000,B 0.000,C 90.000,E1 271.718} C_DIS
LIN {X 0.049,Y -538.745,Z 1042.303,A 0.000,B 0.000,C 90.000,E1 270.573} C_DIS
LIN {X 0.130,Y -537.626,Z 1042.294,A 0.000,B 0.000,C 90.000,E1 268.854} C_DIS
LIN {X 0.190,Y -536.595,Z 1042.286,A 0.000,B 0.000,C 90.000,E1 267.421} C_DIS
LIN {X 0.227,Y -535.595,Z 1042.278,A 0.000,B 0.000,C 90.000,E1 265.988} C_DIS
LIN {X -0.230,Y -534.148,Z 1042.267,A 0.000,B 0.000,C 90.000,E1 264.033} C_DIS
LIN {X -0.152,Y -532.963,Z 1042.259,A 0.000,B 0.000,C 90.000,E1 262.591} C_DIS
LIN {X -0.022,Y -531.424,Z 1042.251,A 0.000,B 0.000,C 90.000,E1 261.141} C_DIS
LIN {X 0.217,Y -528.598,Z 1042.236,A 0.000,B 0.000,C 90.000,E1 258.522} C_DIS
LIN {X -0.130,Y -526.716,Z 1042.227,A 0.000,B 0.000,C 90.000,E1 256.825} C_DIS
LIN {X 0.237,Y -524.844,Z 1042.217,A 0.000,B 0.000,C 90.000,E1 255.046} C_DIS
LIN {X 0.059,Y -522.991,Z 1042.207,A 0.000,B 0.000,C 90.000,E1 253.323} C_DIS
LIN {X -0.001,Y -521.429,Z 1042.199,A 0.000,B 0.000,C 90.000,E1 251.873} C_DIS
LIN {X -0.085,Y -519.673,Z 1042.191,A 0.000,B 0.000,C 90.000,E1 250.423} C_DIS
LIN {X 0.063,Y -517.156,Z 1042.180,A 0.000,B 0.000,C 90.000,E1 248.358} C_DIS
LIN {X 0.121,Y -515.703,Z 1042.173,A 0.000,B 0.000,C 90.000,E1 247.177} C_DIS
LIN {X -0.188,Y -513.638,Z 1042.165,A 0.000,B 0.000,C 90.000,E1 245.741} C_DIS
LIN {X 0.031,Y -511.797,Z 1042.159,A 0.000,B 0.000,C 90.000,E1 244.537} C_DIS
LIN {X 0.094,Y -509.417,Z 1042.150,A 0.000,B 0.000,C 90.000,E1 243.050} C_DIS
LIN {X 0.158,Y -507.947,Z 1042.145,A 0.000,B 0.000,C 90.000,E1 242.153} C_DIS
LIN {X 0.147,Y -505.288,Z 1042.137,A 0.000,B 0.000,C 90.000,E1 240.667} C_DIS
LIN {X 0.198,Y -502.014,Z 1042.127,A 0.000,B 0.000,C 90.000,E1 238.869} C_DIS
LIN {X -0.253,Y -498.667,Z 1042.117,A 0.000,B 0.000,C 90.000,E1 237.120} C_DIS
LIN {X 0.044,Y -496.292,Z 1042.110,A 0.000,B 0.000,C 90.000,E1 235.881} C_DIS
LIN {X -0.246,Y -493.070,Z 1042.102,A 0.000,B 0.000,C 90.000,E1 234.402} C_DIS
LIN {X 0.091,Y -489.586,Z 1042.094,A 0.000,B 0.000,C 90.000,E1 232.844} C_DIS
LIN {X -0.035,Y -485.974,Z 1042.085,A 0.000,B 0.000,C 90.000,E1 231.331} C_DIS
LIN {X 0.069,Y -482.482,Z 1042.077,A 0.000,B 0.000,C 90.000,E1 229.784} C_DIS
LIN {X 0.082,Y -477.198,Z 1042.063,A 0.000,B 0.000,C 90.000,E1 227.310} C_DIS
LIN {X 0.296,Y -474.014,Z 1042.054,A 0.000,B 0.000,C 90.000,E1 225.729} C_DIS
LIN {X 0.110,Y -470.771,Z 1042.046,A 0.000,B 0.000,C 90.000,E1 224.190} C_DIS
LIN {X -0.043,Y -466.969,Z 1042.035,A 0.000,B 0.000,C 90.000,E1 222.324} C_DIS
LIN {X 0.069,Y -463.065,Z 1042.025,A 0.000,B 0.000,C 90.000,E1 220.415} C_DIS
LIN {X 0.045,Y -459.744,Z 1042.016,A 0.000,B 0.000,C 90.000,E1 218.830} C_DIS
LIN {X 0.122,Y -454.920,Z 1042.003,A 0.000,B 0.000,C 90.000,E1 216.583} C_DIS
LIN {X 0.159,Y -450.242,Z 1041.991,A 0.000,B 0.000,C 90.000,E1 214.326} C_DIS
LIN {X -0.128,Y -446.206,Z 1041.980,A 0.000,B 0.000,C 90.000,E1 212.418} C_DIS
LIN {X -0.131,Y -441.862,Z 1041.969,A 0.000,B 0.000,C 90.000,E1 210.463} C_DIS
LIN {X -0.082,Y -437.434,Z 1041.958,A 0.000,B 0.000,C 90.000,E1 208.487} C_DIS
LIN {X -0.140,Y -431.558,Z 1041.944,A 0.000,B 0.000,C 90.000,E1 205.848} C_DIS
LIN {X -0.006,Y -425.262,Z 1041.927,A 0.000,B 0.000,C 90.000,E1 202.823} C_DIS
LIN {X -0.106,Y -422.099,Z 1041.917,A 0.000,B 0.000,C 90.000,E1 201.153} C_DIS
LIN {X -0.063,Y -415.141,Z 1041.893,A 0.000,B 0.000,C 90.000,E1 196.732} C_DIS
LIN {X 0.063,Y -413.081,Z 1041.882,A 0.000,B 0.000,C 90.000,E1 194.662} C_DIS
LIN {X 0.117,Y -412.293,Z 1041.872,A 0.000,B 0.000,C 90.000,E1 192.939} C_DIS
LIN {X 0.184,Y -412.586,Z 1041.868,A 0.000,B 0.000,C 90.000,E1 192.243} C_DIS
LIN {X -0.065,Y -413.453,Z 1041.864,A 0.000,B 0.000,C 90.000,E1 191.591} C_DIS
LIN {X -0.027,Y -414.165,Z 1041.862,A 0.000,B 0.000,C 90.000,E1 191.243} C_DIS
LIN {X 0.073,Y -415.087,Z 1041.861,A 0.000,B 0.000,C 90.000,E1 190.894} C_DIS
LIN {X -0.133,Y -418.344,Z 1041.856,A 0.000,B 0.000,C 90.000,E1 190.074} C_DIS
LIN {X 0.175,Y -422.661,Z 1041.852,A 0.000,B 0.000,C 90.000,E1 189.265} C_DIS
LIN {X 0.136,Y -432.929,Z 1041.843,A 0.000,B 0.000,C 90.000,E1 187.757} C_DIS
LIN {X 0.176,Y -446.027,Z 1041.833,A 0.000,B 0.000,C 90.000,E1 185.967} C_DIS
LIN {X -0.209,Y -451.866,Z 1041.829,A 0.000,B 0.000,C 90.000,E1 185.220} C_DIS
LIN {X -0.087,Y -458.945,Z 1041.824,A 0.000,B 0.000,C 90.000,E1 184.245} C_DIS
LIN {X -0.134,Y -463.515,Z 1041.820,A 0.000,B 0.000,C 90.000,E1 183.612} C_DIS
LIN {X 0.078,Y -470.066,Z 1041.815,A 0.000,B 0.000,C 90.000,E1 182.636} C_DIS
LIN {X 0.223,Y -475.423,Z 1041.810,A 0.000,B 0.000,C 90.000,E1 181.835} C_DIS
LIN {X 0.106,Y -479.288,Z 1041.807,A 0.000,B 0.000,C 90.000,E1 181.260} C_DIS
LIN {X -0.194,Y -480.382,Z 1041.806,A 0.000,B 0.000,C 90.000,E1 181.146} C_DIS
LIN {X -0.086,Y -487.206,Z 1041.800,A 0.000,B 0.000,C 90.000,E1 180.057} C_DIS
LIN {X 0.079,Y -493.961,Z 1041.794,A 0.000,B 0.000,C 90.000,E1 178.969} C_DIS
LIN {X 0.164,Y -499.624,Z 1041.789,A 0.000,B 0.000,C 90.000,E1 178.051} C_DIS
LIN {X 0.010,Y -507.470,Z 1041.782,A 0.000,B 0.000,C 90.000,E1 176.731} C_DIS
LIN {X -0.130,Y -515.180,Z 1041.775,A 0.000,B 0.000,C 90.000,E1 175.412} C_DIS
LIN {X 0.173,Y -523.601,Z 1041.766,A 0.000,B 0.000,C 90.000,E1 173.913} C_DIS
LIN {X 0.119,Y -531.839,Z 1041.758,A 0.000,B 0.000,C 90.000,E1 172.470} C_DIS
LIN {X 0.148,Y -538.197,Z 1041.752,A 0.000,B 0.000,C 90.000,E1 171.319} C_DIS
LIN {X -0.104,Y -544.493,Z 1041.746,A 0.000,B 0.000,C 90.000,E1 170.208} C_DIS
LIN {X -0.249,Y -552.259,Z 1041.738,A 0.000,B 0.000,C 90.000,E1 168.814} C_DIS
LIN {X 0.105,Y -558.965,Z 1041.731,A 0.000,B 0.000,C 90.000,E1 167.521} C_DIS
LIN {X 0.159,Y -564.813,Z 1041.725,A 0.000,B 0.000,C 90.000,E1 166.408} C_DIS
LIN {X -0.124,Y -570.375,Z 1041.719,A 0.000,B 0.000,C 90.000,E1 165.338} C_DIS
LIN {X 0.226,Y -575.772,Z 1041.713,A 0.000,B 0.000,C 90.000,E1 164.212} C_DIS
LIN {X 0.008,Y -581.607,Z 1041.706,A 0.000,B 0.000,C 90.000,E1 163.015} C_DIS
LIN {X 0.203,Y -585.826,Z 1041.700,A 0.000,B 0.000,C 90.000,E1 162.054} C_DIS
LIN {X 0.186,Y -590.406,Z 1041.694,A 0.000,B 0.000,C 90.000,E1 160.986} C_DIS
LIN {X -0.261,Y -595.740,Z 1041.687,A 0.000,B 0.000,C 90.000,E1 159.699} C_DIS
LIN {X 0.250,Y -599.638,Z 1041.681,A 0.000,B 0.000,C 90.000,E1 158.592} C_DIS
LIN {X 0.260,Y -603.305,Z 1041.675,A 0.000,B 0.000,C 90.000,E1 157.539} C_DIS
LIN {X 0.265,Y -607.633,Z 1041.668,A 0.000,B 0.000,C 90.000,E1 156.230} C_DIS
LIN {X -0.177,Y -610.868,Z 1041.662,A 0.000,B 0.000,C 90.000,E1 155.229} C_DIS
LIN {X 0.233,Y -613.790,Z 1041.657,A 0.000,B 0.000,C 90.000,E1 154.152} C_DIS
LIN {X 0.113,Y -617.268,Z 1041.649,A 0.000,B 0.000,C 90.000,E1 152.871} C_DIS
LIN {X 0.053,Y -619.978,Z 1041.644,A 0.000,B 0.000,C 90.000,E1 151.847} C_DIS
LIN {X -0.226,Y -624.435,Z 1041.634,A 0.000,B 0.000,C 90.000,E1 150.078} C_DIS
LIN {X -0.092,Y -628.713,Z 1041.624,A 0.000,B 0.000,C 90.000,E1 148.280} C_DIS
LIN {X 0.089,Y -631.036,Z 1041.618,A 0.000,B 0.000,C 90.000,E1 147.248} C_DIS
LIN {X -0.202,Y -633.970,Z 1041.611,A 0.000,B 0.000,C 90.000,E1 146.008} C_DIS
LIN {X -0.067,Y -637.362,Z 1041.603,A 0.000,B 0.000,C 90.000,E1 144.482} C_DIS
LIN {X -0.290,Y -639.659,Z 1041.597,A 0.000,B 0.000,C 90.000,E1 143.497} C_DIS
LIN {X 0.221,Y -643.629,Z 1041.587,A 0.000,B 0.000,C 90.000,E1 141.698} C_DIS
LIN {X -0.185,Y -647.612,Z 1041.578,A 0.000,B 0.000,C 90.000,E1 139.989} C_DIS
LIN {X 0.039,Y -649.814,Z 1041.572,A 0.000,B 0.000,C 90.000,E1 138.976} C_DIS
LIN {X -0.182,Y -652.613,Z 1041.565,A 0.000,B 0.000,C 90.000,E1 137.757} C_DIS
LIN {X -0.008,Y -657.382,Z 1041.554,A 0.000,B 0.000,C 90.000,E1 135.769} C_DIS
LIN {X -0.231,Y -664.690,Z 1041.539,A 0.000,B 0.000,C 90.000,E1 133.095} C_DIS
LIN {X -0.209,Y -670.124,Z 1041.529,A 0.000,B 0.000,C 90.000,E1 131.148} C_DIS
LIN {X 0.420,Y -674.146,Z 1041.521,A 0.000,B 0.000,C 90.000,E1 129.644} C_DIS
LIN {X 0.140,Y -676.812,Z 1041.515,A 0.000,B 0.000,C 90.000,E1 128.705} C_DIS
LIN {X -0.234,Y -678.717,Z 1041.511,A 0.000,B 0.000,C 90.000,E1 128.016} C_DIS
LIN {X 0.103,Y -681.770,Z 1041.505,A 0.000,B 0.000,C 90.000,E1 126.790} C_DIS
LIN {X 0.289,Y -686.082,Z 1041.495,A 0.000,B 0.000,C 90.000,E1 125.105} C_DIS
LIN {X 0.188,Y -690.326,Z 1041.486,A 0.000,B 0.000,C 90.000,E1 123.452} C_DIS
LIN {X -0.058,Y -693.749,Z 1041.478,A 0.000,B 0.000,C 90.000,E1 122.054} C_DIS
LIN {X -0.045,Y -696.460,Z 1041.472,A 0.000,B 0.000,C 90.000,E1 120.875} C_DIS
LIN {X 0.117,Y -698.269,Z 1041.466,A 0.000,B 0.000,C 90.000,E1 119.922} C_DIS
LIN {X 0.291,Y -699.362,Z 1041.462,A 0.000,B 0.000,C 90.000,E1 119.205} C_DIS
LIN {X 0.131,Y -700.579,Z 1041.457,A 0.000,B 0.000,C 90.000,E1 118.281} C_DIS
LIN {X 0.207,Y -702.188,Z 1041.449,A 0.000,B 0.000,C 90.000,E1 116.873} C_DIS
LIN {X -0.245,Y -703.156,Z 1041.444,A 0.000,B 0.000,C 90.000,E1 115.976} C_DIS
LIN {X -0.053,Y -703.867,Z 1041.439,A 0.000,B 0.000,C 90.000,E1 115.027} C_DIS
LIN {X 0.230,Y -704.024,Z 1041.438,A 0.000,B 0.000,C 90.000,E1 114.771} C_DIS
LIN {X -0.135,Y -703.979,Z 1041.435,A 0.000,B 0.000,C 90.000,E1 114.335} C_DIS
LIN {X 0.148,Y -703.895,Z 1041.434,A 0.000,B 0.000,C 90.000,E1 114.079} C_DIS
LIN {X -0.216,Y -702.892,Z 1041.431,A 0.000,B 0.000,C 90.000,E1 113.643} C_DIS
LIN {X 0.062,Y -702.243,Z 1041.430,A 0.000,B 0.000,C 90.000,E1 113.387} C_DIS
LIN {X -0.179,Y -698.714,Z 1041.427,A 0.000,B 0.000,C 90.000,E1 112.823} C_DIS
LIN {X -0.048,Y -697.672,Z 1041.426,A 0.000,B 0.000,C 90.000,E1 112.695} C_DIS
LIN {X -0.186,Y -696.095,Z 1041.425,A 0.000,B 0.000,C 90.000,E1 112.589} C_DIS
LIN {X 0.048,Y -689.154,Z 1041.423,A 0.000,B 0.000,C 90.000,E1 112.206} C_DIS
LIN {X -0.270,Y -687.109,Z 1041.423,A 0.000,B 0.000,C 90.000,E1 112.153} C_DIS
LIN {X -0.153,Y -685.087,Z 1041.423,A 0.000,B 0.000,C 90.000,E1 112.078} C_DIS
LIN {X 0.093,Y -683.572,Z 1041.422,A 0.000,B 0.000,C 90.000,E1 112.025} C_DIS
LIN {X -0.170,Y -675.414,Z 1041.422,A 0.000,B 0.000,C 90.000,E1 111.950} C_DIS
LIN {X 0.365,Y -611.182,Z 1041.422,A 0.000,B 0.000,C 90.000,E1 111.897} C_DIS
LIN {X 0.119,Y -603.804,Z 1041.420,A 0.000,B 0.000,C 90.000,E1 111.663} C_DIS
LIN {X 0.050,Y -597.652,Z 1041.419,A 0.000,B 0.000,C 90.000,E1 111.354} C_DIS
LIN {X 0.104,Y -592.014,Z 1041.417,A 0.000,B 0.000,C 90.000,E1 110.972} C_DIS
LIN {X -0.145,Y -583.928,Z 1041.413,A 0.000,B 0.000,C 90.000,E1 110.355} C_DIS
LIN {X 0.309,Y -575.775,Z 1041.409,A 0.000,B 0.000,C 90.000,E1 109.631} C_DIS
LIN {X 0.018,Y -569.735,Z 1041.407,A 0.000,B 0.000,C 90.000,E1 109.214} C_DIS
LIN {X 0.053,Y -561.454,Z 1041.404,A 0.000,B 0.000,C 90.000,E1 108.725} C_DIS
LIN {X 0.112,Y -554.830,Z 1041.402,A 0.000,B 0.000,C 90.000,E1 108.362} C_DIS
LIN {X 0.234,Y -549.456,Z 1041.400,A 0.000,B 0.000,C 90.000,E1 108.000} C_DIS
LIN {X 0.192,Y -547.957,Z 1041.399,A 0.000,B 0.000,C 90.000,E1 107.819} C_DIS
LIN {X 0.150,Y -547.935,Z 1041.399,A 0.000,B 0.000,C 90.000,E1 107.819} C_DIS
LIN {X -0.242,Y -547.499,Z 1041.398,A 0.000,B 0.000,C 90.000,E1 107.583} C_DIS
LIN {X -0.110,Y -547.578,Z 1041.394,A 0.000,B 0.000,C 90.000,E1 106.985} C_DIS
LIN {X -0.054,Y -548.130,Z 1041.390,A 0.000,B 0.000,C 90.000,E1 106.134} C_DIS
LIN {X -0.145,Y -549.238,Z 1041.379,A 0.000,B 0.000,C 90.000,E1 104.175} C_DIS
LIN {X 0.110,Y -551.921,Z 1041.360,A 0.000,B 0.000,C 90.000,E1 100.782} C_DIS
LIN {X -0.114,Y -554.321,Z 1041.348,A 0.000,B 0.000,C 90.000,E1 98.568} C_DIS
LIN {X -0.076,Y -556.258,Z 1041.338,A 0.000,B 0.000,C 90.000,E1 96.891} C_DIS
LIN {X -0.258,Y -557.481,Z 1041.332,A 0.000,B 0.000,C 90.000,E1 95.796} C_DIS
LIN {X 0.133,Y -558.473,Z 1041.326,A 0.000,B 0.000,C 90.000,E1 94.645} C_DIS
LIN {X 0.022,Y -559.478,Z 1041.318,A 0.000,B 0.000,C 90.000,E1 93.269} C_DIS
LIN {X 0.047,Y -560.316,Z 1041.309,A 0.000,B 0.000,C 90.000,E1 91.604} C_DIS
LIN {X 0.051,Y -560.914,Z 1041.300,A 0.000,B 0.000,C 90.000,E1 89.943} C_DIS
LIN {X 0.067,Y -561.451,Z 1041.291,A 0.000,B 0.000,C 90.000,E1 88.282} C_DIS
LIN {X 0.006,Y -561.906,Z 1041.283,A 0.000,B 0.000,C 90.000,E1 86.906} C_DIS
LIN {X 0.080,Y -562.498,Z 1041.274,A 0.000,B 0.000,C 90.000,E1 85.241} C_DIS
LIN {X 0.129,Y -562.868,Z 1041.266,A 0.000,B 0.000,C 90.000,E1 83.856} C_DIS
LIN {X 0.030,Y -563.393,Z 1041.254,A 0.000,B 0.000,C 90.000,E1 81.659} C_DIS
LIN {X 0.190,Y -564.261,Z 1041.240,A 0.000,B 0.000,C 90.000,E1 79.162} C_DIS
LIN {X -0.134,Y -565.292,Z 1041.228,A 0.000,B 0.000,C 90.000,E1 76.992} C_DIS
LIN {X -0.089,Y -566.291,Z 1041.219,A 0.000,B 0.000,C 90.000,E1 75.338} C_DIS
LIN {X 0.077,Y -568.094,Z 1041.205,A 0.000,B 0.000,C 90.000,E1 72.851} C_DIS
LIN {X -0.016,Y -569.004,Z 1041.199,A 0.000,B 0.000,C 90.000,E1 71.764} C_DIS
LIN {X 0.061,Y -570.355,Z 1041.190,A 0.000,B 0.000,C 90.000,E1 70.115} C_DIS
LIN {X -0.001,Y -571.118,Z 1041.184,A 0.000,B 0.000,C 90.000,E1 69.028} C_DIS
LIN {X -0.030,Y -572.126,Z 1041.176,A 0.000,B 0.000,C 90.000,E1 67.667} C_DIS
LIN {X -0.208,Y -573.133,Z 1041.167,A 0.000,B 0.000,C 90.000,E1 66.049} C_DIS
LIN {X -0.133,Y -574.048,Z 1041.158,A 0.000,B 0.000,C 90.000,E1 64.409} C_DIS
LIN {X 0.053,Y -574.994,Z 1041.147,A 0.000,B 0.000,C 90.000,E1 62.487} C_DIS
LIN {X 0.178,Y -575.653,Z 1041.138,A 0.000,B 0.000,C 90.000,E1 60.845} C_DIS
LIN {X 0.159,Y -576.502,Z 1041.128,A 0.000,B 0.000,C 90.000,E1 58.948} C_DIS
LIN {X 0.107,Y -577.094,Z 1041.119,A 0.000,B 0.000,C 90.000,E1 57.327} C_DIS
LIN {X -0.252,Y -577.446,Z 1041.111,A 0.000,B 0.000,C 90.000,E1 56.008} C_DIS
LIN {X 0.047,Y -577.633,Z 1041.105,A 0.000,B 0.000,C 90.000,E1 54.895} C_DIS
LIN {X -0.123,Y -577.795,Z 1041.099,A 0.000,B 0.000,C 90.000,E1 53.829} C_DIS
LIN {X 0.170,Y -577.763,Z 1041.093,A 0.000,B 0.000,C 90.000,E1 52.718} C_DIS
LIN {X 0.030,Y -577.719,Z 1041.090,A 0.000,B 0.000,C 90.000,E1 52.190} C_DIS
LIN {X 0.053,Y -577.523,Z 1041.085,A 0.000,B 0.000,C 90.000,E1 51.376} C_DIS
LIN {X 0.096,Y -576.787,Z 1041.076,A 0.000,B 0.000,C 90.000,E1 49.747} C_DIS
LIN {X -0.034,Y -576.041,Z 1041.069,A 0.000,B 0.000,C 90.000,E1 48.405} C_DIS
LIN {X 0.060,Y -575.259,Z 1041.063,A 0.000,B 0.000,C 90.000,E1 47.310} C_DIS
LIN {X 0.014,Y -574.570,Z 1041.058,A 0.000,B 0.000,C 90.000,E1 46.500} C_DIS
LIN {X -0.023,Y -573.709,Z 1041.054,A 0.000,B 0.000,C 90.000,E1 45.688} C_DIS
LIN {X 0.027,Y -572.216,Z 1041.048,A 0.000,B 0.000,C 90.000,E1 44.595} C_DIS
LIN {X -0.048,Y -570.955,Z 1041.043,A 0.000,B 0.000,C 90.000,E1 43.785} C_DIS
LIN {X -0.026,Y -569.091,Z 1041.037,A 0.000,B 0.000,C 90.000,E1 42.690} C_DIS
LIN {X 0.278,Y -567.487,Z 1041.033,A 0.000,B 0.000,C 90.000,E1 41.838} C_DIS
LIN {X -0.236,Y -565.628,Z 1041.028,A 0.000,B 0.000,C 90.000,E1 41.067} C_DIS
LIN {X -0.018,Y -564.348,Z 1041.025,A 0.000,B 0.000,C 90.000,E1 40.496} C_DIS
LIN {X 0.229,Y -562.120,Z 1041.020,A 0.000,B 0.000,C 90.000,E1 39.644} C_DIS
LIN {X -0.006,Y -560.538,Z 1041.017,A 0.000,B 0.000,C 90.000,E1 39.116} C_DIS
LIN {X -0.165,Y -557.841,Z 1041.013,A 0.000,B 0.000,C 90.000,E1 38.302} C_DIS
LIN {X 0.007,Y -555.876,Z 1041.010,A 0.000,B 0.000,C 90.000,E1 37.729} C_DIS
LIN {X 0.238,Y -552.673,Z 1041.005,A 0.000,B 0.000,C 90.000,E1 36.870} C_DIS
LIN {X -0.071,Y -550.362,Z 1041.002,A 0.000,B 0.000,C 90.000,E1 36.343} C_DIS
LIN {X -0.092,Y -547.204,Z 1040.998,A 0.000,B 0.000,C 90.000,E1 35.644} C_DIS
LIN {X -0.281,Y -543.134,Z 1040.993,A 0.000,B 0.000,C 90.000,E1 34.818} C_DIS
LIN {X 0.243,Y -538.794,Z 1040.989,A 0.000,B 0.000,C 90.000,E1 33.913} C_DIS
LIN {X -0.180,Y -533.412,Z 1040.983,A 0.000,B 0.000,C 90.000,E1 32.959} C_DIS
LIN {X 0.092,Y -529.154,Z 1040.979,A 0.000,B 0.000,C 90.000,E1 32.212} C_DIS
LIN {X 0.004,Y -522.848,Z 1040.973,A 0.000,B 0.000,C 90.000,E1 31.209} C_DIS
LIN {X -0.164,Y -515.739,Z 1040.968,A 0.000,B 0.000,C 90.000,E1 30.207} C_DIS
LIN {X -0.067,Y -510.273,Z 1040.964,A 0.000,B 0.000,C 90.000,E1 29.461} C_DIS
LIN {X -0.091,Y -505.507,Z 1040.960,A 0.000,B 0.000,C 90.000,E1 28.871} C_DIS
LIN {X 0.037,Y -501.749,Z 1040.958,A 0.000,B 0.000,C 90.000,E1 28.409} C_DIS
LIN {X -0.095,Y -495.018,Z 1040.954,A 0.000,B 0.000,C 90.000,E1 27.692} C_DIS
LIN {X -0.220,Y -489.514,Z 1040.951,A 0.000,B 0.000,C 90.000,E1 27.129} C_DIS
LIN {X 0.092,Y -485.286,Z 1040.948,A 0.000,B 0.000,C 90.000,E1 26.668} C_DIS
LIN {X -0.111,Y -475.290,Z 1040.943,A 0.000,B 0.000,C 90.000,E1 25.720} C_DIS
LIN {X 0.013,Y -465.196,Z 1040.938,A 0.000,B 0.000,C 90.000,E1 24.771} C_DIS
LIN {X -0.226,Y -453.186,Z 1040.932,A 0.000,B 0.000,C 90.000,E1 23.770} C_DIS
LIN {X 0.024,Y -432.083,Z 1040.922,A 0.000,B 0.000,C 90.000,E1 21.897} C_DIS
LIN {X 0.086,Y -418.870,Z 1040.915,A 0.000,B 0.000,C 90.000,E1 20.610} C_DIS
LIN {X -0.119,Y -404.705,Z 1040.906,A 0.000,B 0.000,C 90.000,E1 19.087} C_DIS
LIN {X -0.158,Y -400.631,Z 1040.903,A 0.000,B 0.000,C 90.000,E1 18.598} C_DIS
LIN {X 0.031,Y -396.838,Z 1040.900,A 0.000,B 0.000,C 90.000,E1 18.055} C_DIS
LIN {X 0.028,Y -394.366,Z 1040.898,A 0.000,B 0.000,C 90.000,E1 17.638} C_DIS
LIN {X 0.138,Y -392.174,Z 1040.895,A 0.000,B 0.000,C 90.000,E1 17.040} C_DIS
LIN {X 0.054,Y -391.341,Z 1040.891,A 0.000,B 0.000,C 90.000,E1 16.386} C_DIS
LIN {X 0.123,Y -391.385,Z 1040.888,A 0.000,B 0.000,C 90.000,E1 15.843} C_DIS
LIN {X 0.151,Y -392.301,Z 1040.882,A 0.000,B 0.000,C 90.000,E1 14.773} C_DIS
LIN {X -0.002,Y -398.283,Z 1040.857,A 0.000,B 0.000,C 90.000,E1 10.197} C_DIS
LIN {X -0.178,Y -405.265,Z 1040.835,A 0.000,B 0.000,C 90.000,E1 6.372} C_DIS
LIN {X 0.171,Y -408.972,Z 1040.826,A 0.000,B 0.000,C 90.000,E1 4.588} C_DIS
LIN {X 0.142,Y -412.070,Z 1040.818,A 0.000,B 0.000,C 90.000,E1 3.212} C_DIS
LIN {X 0.159,Y -413.909,Z 1040.815,A 0.000,B 0.000,C 90.000,E1 2.694} C_DIS
LIN {X 0.158,Y -414.666,Z 1040.814,A 0.000,B 0.000,C 90.000,E1 2.522} C_DIS
LIN {X -0.185,Y -417.785,Z 1040.811,A 0.000,B 0.000,C 90.000,E1 2.064} C_DIS
LIN {X 0.022,Y -422.580,Z 1040.809,A 0.000,B 0.000,C 90.000,E1 1.547} C_DIS
LIN {X 0.212,Y -439.268,Z 1040.803,A 0.000,B 0.000,C 90.000,E1 0.458} C_DIS
LIN {X 0.119,Y -456.981,Z 1040.797,A 0.000,B 0.000,C 90.000,E1 359.370} C_DIS
LIN {X -0.111,Y -473.550,Z 1040.791,A 0.000,B 0.000,C 90.000,E1 358.396} C_DIS
LIN {X 0.088,Y -486.407,Z 1040.787,A 0.000,B 0.000,C 90.000,E1 357.593} C_DIS
LIN {X 0.023,Y -497.694,Z 1040.783,A 0.000,B 0.000,C 90.000,E1 356.906} C_DIS
LIN {X 0.194,Y -505.246,Z 1040.780,A 0.000,B 0.000,C 90.000,E1 356.388} C_DIS
LIN {X 0.057,Y -516.090,Z 1040.776,A 0.000,B 0.000,C 90.000,E1 355.641} C_DIS
LIN {X 0.019,Y -524.859,Z 1040.772,A 0.000,B 0.000,C 90.000,E1 354.951} C_DIS
LIN {X -0.250,Y -531.915,Z 1040.769,A 0.000,B 0.000,C 90.000,E1 354.375} C_DIS
LIN {X 0.190,Y -538.670,Z 1040.765,A 0.000,B 0.000,C 90.000,E1 353.685} C_DIS
LIN {X -0.139,Y -545.029,Z 1040.761,A 0.000,B 0.000,C 90.000,E1 353.053} C_DIS
LIN {X 0.044,Y -549.974,Z 1040.758,A 0.000,B 0.000,C 90.000,E1 352.470} C_DIS
LIN {X -0.072,Y -555.485,Z 1040.754,A 0.000,B 0.000,C 90.000,E1 351.781} C_DIS
LIN {X 0.184,Y -559.438,Z 1040.751,A 0.000,B 0.000,C 90.000,E1 351.197} C_DIS
LIN {X 0.232,Y -563.894,Z 1040.747,A 0.000,B 0.000,C 90.000,E1 350.500} C_DIS
LIN {X 0.077,Y -568.742,Z 1040.743,A 0.000,B 0.000,C 90.000,E1 349.690} C_DIS
LIN {X -0.167,Y -573.912,Z 1040.738,A 0.000,B 0.000,C 90.000,E1 348.757} C_DIS
LIN {X -0.118,Y -577.937,Z 1040.733,A 0.000,B 0.000,C 90.000,E1 347.937} C_DIS
LIN {X -0.132,Y -582.172,Z 1040.728,A 0.000,B 0.000,C 90.000,E1 346.992} C_DIS
LIN {X 0.239,Y -586.707,Z 1040.722,A 0.000,B 0.000,C 90.000,E1 345.880} C_DIS
LIN {X 0.247,Y -591.003,Z 1040.716,A 0.000,B 0.000,C 90.000,E1 344.810} C_DIS
LIN {X -0.255,Y -595.169,Z 1040.710,A 0.000,B 0.000,C 90.000,E1 343.795} C_DIS
LIN {X -0.133,Y -599.103,Z 1040.704,A 0.000,B 0.000,C 90.000,E1 342.725} C_DIS
LIN {X 0.222,Y -602.817,Z 1040.698,A 0.000,B 0.000,C 90.000,E1 341.638} C_DIS
LIN {X 0.140,Y -605.439,Z 1040.694,A 0.000,B 0.000,C 90.000,E1 340.859} C_DIS
LIN {X 0.008,Y -608.646,Z 1040.688,A 0.000,B 0.000,C 90.000,E1 339.826} C_DIS
LIN {X 0.134,Y -611.637,Z 1040.682,A 0.000,B 0.000,C 90.000,E1 338.773} C_DIS
LIN {X 0.078,Y -614.397,Z 1040.676,A 0.000,B 0.000,C 90.000,E1 337.741} C_DIS
LIN {X -0.283,Y -616.938,Z 1040.671,A 0.000,B 0.000,C 90.000,E1 336.741} C_DIS
LIN {X 0.209,Y -619.327,Z 1040.665,A 0.000,B 0.000,C 90.000,E1 335.665} C_DIS
LIN {X -0.080,Y -620.873,Z 1040.661,A 0.000,B 0.000,C 90.000,E1 334.921} C_DIS
LIN {X -0.089,Y -623.348,Z 1040.654,A 0.000,B 0.000,C 90.000,E1 333.640} C_DIS
LIN {X -0.046,Y -625.818,Z 1040.645,A 0.000,B 0.000,C 90.000,E1 332.103} C_DIS
LIN {X 0.304,Y -627.276,Z 1040.639,A 0.000,B 0.000,C 90.000,E1 331.051} C_DIS
LIN {X 0.150,Y -628.876,Z 1040.632,A 0.000,B 0.000,C 90.000,E1 329.793} C_DIS
LIN {X 0.020,Y -630.070,Z 1040.625,A 0.000,B 0.000,C 90.000,E1 328.535} C_DIS
LIN {X 0.235,Y -631.091,Z 1040.618,A 0.000,B 0.000,C 90.000,E1 327.248} C_DIS
LIN {X -0.063,Y -631.760,Z 1040.611,A 0.000,B 0.000,C 90.000,E1 326.008} C_DIS
LIN {X -0.353,Y -632.035,Z 1040.604,A 0.000,B 0.000,C 90.000,E1 324.769} C_DIS
LIN {X 0.088,Y -632.148,Z 1040.596,A 0.000,B 0.000,C 90.000,E1 323.210} C_DIS
LIN {X 0.023,Y -632.281,Z 1040.587,A 0.000,B 0.000,C 90.000,E1 321.698} C_DIS
LIN {X -0.014,Y -632.476,Z 1040.580,A 0.000,B 0.000,C 90.000,E1 320.436} C_DIS
LIN {X -0.050,Y -632.683,Z 1040.573,A 0.000,B 0.000,C 90.000,E1 319.175} C_DIS
LIN {X -0.142,Y -632.800,Z 1040.566,A 0.000,B 0.000,C 90.000,E1 317.919} C_DIS
LIN {X -0.087,Y -633.031,Z 1040.555,A 0.000,B 0.000,C 90.000,E1 315.891} C_DIS
LIN {X 0.170,Y -633.285,Z 1040.547,A 0.000,B 0.000,C 90.000,E1 314.352} C_DIS
LIN {X 0.097,Y -633.537,Z 1040.540,A 0.000,B 0.000,C 90.000,E1 313.095} C_DIS
LIN {X 0.136,Y -633.693,Z 1040.534,A 0.000,B 0.000,C 90.000,E1 312.081} C_DIS
LIN {X 0.060,Y -633.816,Z 1040.527,A 0.000,B 0.000,C 90.000,E1 310.825} C_DIS
LIN {X 0.162,Y -633.877,Z 1040.521,A 0.000,B 0.000,C 90.000,E1 309.806} C_DIS
LIN {X -0.218,Y -633.865,Z 1040.516,A 0.000,B 0.000,C 90.000,E1 308.830} C_DIS
LIN {X 0.135,Y -633.854,Z 1040.506,A 0.000,B 0.000,C 90.000,E1 307.030} C_DIS
LIN {X -0.267,Y -633.957,Z 1040.499,A 0.000,B 0.000,C 90.000,E1 305.804} C_DIS
LIN {X -0.041,Y -634.824,Z 1040.483,A 0.000,B 0.000,C 90.000,E1 303.007} C_DIS
LIN {X -0.187,Y -635.873,Z 1040.472,A 0.000,B 0.000,C 90.000,E1 301.003} C_DIS
LIN {X 0.257,Y -637.285,Z 1040.461,A 0.000,B 0.000,C 90.000,E1 298.949} C_DIS
LIN {X -0.042,Y -638.285,Z 1040.454,A 0.000,B 0.000,C 90.000,E1 297.719} C_DIS
LIN {X 0.188,Y -639.043,Z 1040.448,A 0.000,B 0.000,C 90.000,E1 296.693} C_DIS
LIN {X -0.206,Y -639.476,Z 1040.444,A 0.000,B 0.000,C 90.000,E1 295.976} C_DIS
LIN {X -0.028,Y -639.660,Z 1040.440,A 0.000,B 0.000,C 90.000,E1 295.207} C_DIS
LIN {X -0.059,Y -639.722,Z 1040.434,A 0.000,B 0.000,C 90.000,E1 294.207} C_DIS
LIN {X -0.142,Y -639.531,Z 1040.430,A 0.000,B 0.000,C 90.000,E1 293.462} C_DIS
LIN {X -0.170,Y -639.060,Z 1040.425,A 0.000,B 0.000,C 90.000,E1 292.461} C_DIS
LIN {X -0.259,Y -638.434,Z 1040.421,A 0.000,B 0.000,C 90.000,E1 291.716} C_DIS
LIN {X 0.195,Y -637.584,Z 1040.418,A 0.000,B 0.000,C 90.000,E1 291.173} C_DIS
LIN {X 0.236,Y -636.961,Z 1040.416,A 0.000,B 0.000,C 90.000,E1 290.918} C_DIS
LIN {X 0.088,Y -635.276,Z 1040.414,A 0.000,B 0.000,C 90.000,E1 290.429} C_DIS
LIN {X -0.073,Y -631.997,Z 1040.411,A 0.000,B 0.000,C 90.000,E1 289.939} C_DIS
LIN {X -0.064,Y -631.102,Z 1040.410,A 0.000,B 0.000,C 90.000,E1 289.812} C_DIS
LIN {X -0.256,Y -628.527,Z 1040.409,A 0.000,B 0.000,C 90.000,E1 289.577} C_DIS
LIN {X -0.138,Y -625.689,Z 1040.407,A 0.000,B 0.000,C 90.000,E1 289.322} C_DIS
LIN {X -0.238,Y -624.106,Z 1040.407,A 0.000,B 0.000,C 90.000,E1 289.214} C_DIS
LIN {X 0.210,Y -620.006,Z 1040.406,A 0.000,B 0.000,C 90.000,E1 288.960} C_DIS
LIN {X 0.014,Y -616.785,Z 1040.404,A 0.000,B 0.000,C 90.000,E1 288.779} C_DIS
LIN {X 0.166,Y -614.902,Z 1040.404,A 0.000,B 0.000,C 90.000,E1 288.671} C_DIS
LIN {X 0.153,Y -605.638,Z 1040.402,A 0.000,B 0.000,C 90.000,E1 288.308} C_DIS
LIN {X 0.037,Y -596.747,Z 1040.400,A 0.000,B 0.000,C 90.000,E1 288.000} C_DIS
LIN {X 0.072,Y -589.644,Z 1040.399,A 0.000,B 0.000,C 90.000,E1 287.764} C_DIS
LIN {X -0.050,Y -579.153,Z 1040.397,A 0.000,B 0.000,C 90.000,E1 287.457} C_DIS
LIN {X 0.196,Y -569.482,Z 1040.395,A 0.000,B 0.000,C 90.000,E1 287.094} C_DIS
LIN {X 0.168,Y -566.581,Z 1040.395,A 0.000,B 0.000,C 90.000,E1 286.985} C_DIS
LIN {X 0.060,Y -560.767,Z 1040.393,A 0.000,B 0.000,C 90.000,E1 286.732} C_DIS
LIN {X -0.104,Y -556.480,Z 1040.392,A 0.000,B 0.000,C 90.000,E1 286.496} C_DIS
LIN {X 0.184,Y -554.067,Z 1040.390,A 0.000,B 0.000,C 90.000,E1 286.150} C_DIS
LIN {X -0.120,Y -552.254,Z 1040.387,A 0.000,B 0.000,C 90.000,E1 285.662} C_DIS
LIN {X -0.235,Y -552.115,Z 1040.387,A 0.000,B 0.000,C 90.000,E1 285.607} C_DIS
LIN {X -0.283,Y -585.882,Z 1040.387,A 0.000,B 0.000,C 90.000,E1 285.607} C_DIS
LIN {X -0.037,Y -589.381,Z 1040.386,A 0.000,B 0.000,C 90.000,E1 285.552} C_DIS
LIN {X -0.201,Y -591.534,Z 1040.386,A 0.000,B 0.000,C 90.000,E1 285.536} C_DIS
LIN {X -0.105,Y -596.781,Z 1040.384,A 0.000,B 0.000,C 90.000,E1 285.190} C_DIS
LIN {X 0.164,Y -598.068,Z 1040.384,A 0.000,B 0.000,C 90.000,E1 285.064} C_DIS
LIN {X 0.017,Y -602.066,Z 1040.381,A 0.000,B 0.000,C 90.000,E1 284.592} C_DIS
LIN {X -0.198,Y -603.025,Z 1040.380,A 0.000,B 0.000,C 90.000,E1 284.481} C_DIS
LIN {X -0.014,Y -605.763,Z 1040.377,A 0.000,B 0.000,C 90.000,E1 283.939} C_DIS
LIN {X 0.103,Y -607.358,Z 1040.375,A 0.000,B 0.000,C 90.000,E1 283.536} C_DIS
LIN {X -0.161,Y -608.263,Z 1040.374,A 0.000,B 0.000,C 90.000,E1 283.300} C_DIS
LIN {X 0.172,Y -608.833,Z 1040.372,A 0.000,B 0.000,C 90.000,E1 283.008} C_DIS
LIN {X 0.253,Y -609.824,Z 1040.370,A 0.000,B 0.000,C 90.000,E1 282.479} C_DIS
LIN {X -0.255,Y -610.142,Z 1040.367,A 0.000,B 0.000,C 90.000,E1 282.007} C_DIS
LIN {X -0.165,Y -609.378,Z 1040.364,A 0.000,B 0.000,C 90.000,E1 281.478} C_DIS
LIN {X 0.177,Y -608.785,Z 1040.362,A 0.000,B 0.000,C 90.000,E1 281.186} C_DIS
LIN {X 0.256,Y -607.032,Z 1040.359,A 0.000,B 0.000,C 90.000,E1 280.658} C_DIS
LIN {X 0.212,Y -604.203,Z 1040.356,A 0.000,B 0.000,C 90.000,E1 280.141} C_DIS
LIN {X 0.254,Y -600.570,Z 1040.354,A 0.000,B 0.000,C 90.000,E1 279.613} C_DIS
LIN {X -0.032,Y -598.219,Z 1040.352,A 0.000,B 0.000,C 90.000,E1 279.378} C_DIS
LIN {X 0.170,Y -595.565,Z 1040.351,A 0.000,B 0.000,C 90.000,E1 279.095} C_DIS
LIN {X -0.005,Y -589.885,Z 1040.348,A 0.000,B 0.000,C 90.000,E1 278.624} C_DIS
LIN {X 0.298,Y -583.551,Z 1040.346,A 0.000,B 0.000,C 90.000,E1 278.163} C_DIS
LIN {X -0.160,Y -581.540,Z 1040.345,A 0.000,B 0.000,C 90.000,E1 278.106} C_DIS
LIN {X -0.172,Y -577.077,Z 1040.344,A 0.000,B 0.000,C 90.000,E1 277.936} C_DIS
LIN {X 0.125,Y -576.067,Z 1040.344,A 0.000,B 0.000,C 90.000,E1 277.871} C_DIS
LIN {X -0.024,Y -569.321,Z 1040.344,A 0.000,B 0.000,C 90.000,E1 277.814} C_DIS
LIN {X -0.073,Y -545.797,Z 1040.343,A 0.000,B 0.000,C 90.000,E1 277.814} C_DIS
LIN {X 0.229,Y -546.035,Z 1040.342,A 0.000,B 0.000,C 90.000,E1 277.587} C_DIS
LIN {X 0.108,Y -545.814,Z 1040.341,A 0.000,B 0.000,C 90.000,E1 277.409} C_DIS
LIN {X -0.154,Y -545.315,Z 1040.340,A 0.000,B 0.000,C 90.000,E1 277.296} C_DIS
LIN {X 0.127,Y -544.478,Z 1040.340,A 0.000,B 0.000,C 90.000,E1 277.125} C_DIS
LIN {X 0.263,Y -543.124,Z 1040.339,A 0.000,B 0.000,C 90.000,E1 276.947} C_DIS
LIN {X 0.221,Y -543.101,Z 1040.339,A 0.000,B 0.000,C 90.000,E1 276.947} C_DIS
LIN {X 0.076,Y -540.880,Z 1040.322,A 0.000,B 0.000,C 90.000,E1 274.012} C_DIS
LIN {X 0.263,Y -539.598,Z 1040.310,A 0.000,B 0.000,C 90.000,E1 271.718} C_DIS
LIN {X -0.209,Y -538.979,Z 1040.303,A 0.000,B 0.000,C 90.000,E1 270.630} C_DIS
LIN {X -0.123,Y -537.849,Z 1040.294,A 0.000,B 0.000,C 90.000,E1 268.912} C_DIS
LIN {X -0.049,Y -536.395,Z 1040.283,A 0.000,B 0.000,C 90.000,E1 266.906} C_DIS
LIN {X 0.018,Y -535.368,Z 1040.275,A 0.000,B 0.000,C 90.000,E1 265.469} C_DIS
LIN {X 0.106,Y -534.129,Z 1040.265,A 0.000,B 0.000,C 90.000,E1 263.742} C_DIS
LIN {X 0.147,Y -533.167,Z 1040.259,A 0.000,B 0.000,C 90.000,E1 262.591} C_DIS
LIN {X -0.246,Y -531.674,Z 1040.251,A 0.000,B 0.000,C 90.000,E1 261.197} C_DIS
LIN {X -0.026,Y -529.130,Z 1040.238,A 0.000,B 0.000,C 90.000,E1 258.870} C_DIS
LIN {X 0.158,Y -527.267,Z 1040.229,A 0.000,B 0.000,C 90.000,E1 257.117} C_DIS
LIN {X 0.046,Y -525.069,Z 1040.217,A 0.000,B 0.000,C 90.000,E1 255.102} C_DIS
LIN {X -0.123,Y -522.890,Z 1040.206,A 0.000,B 0.000,C 90.000,E1 253.087} C_DIS
LIN {X -0.186,Y -521.286,Z 1040.198,A 0.000,B 0.000,C 90.000,E1 251.638} C_DIS
LIN {X -0.277,Y -519.498,Z 1040.190,A 0.000,B 0.000,C 90.000,E1 250.188} C_DIS
LIN {X -0.089,Y -517.362,Z 1040.180,A 0.000,B 0.000,C 90.000,E1 248.411} C_DIS
LIN {X -0.022,Y -515.896,Z 1040.174,A 0.000,B 0.000,C 90.000,E1 247.230} C_DIS
LIN {X 0.147,Y -513.879,Z 1040.165,A 0.000,B 0.000,C 90.000,E1 245.741} C_DIS
LIN {X 0.018,Y -511.519,Z 1040.157,A 0.000,B 0.000,C 90.000,E1 244.280} C_DIS
LIN {X -0.252,Y -509.634,Z 1040.151,A 0.000,B 0.000,C 90.000,E1 243.127} C_DIS
LIN {X 0.137,Y -507.627,Z 1040.144,A 0.000,B 0.000,C 90.000,E1 241.897} C_DIS
LIN {X 0.117,Y -504.966,Z 1040.136,A 0.000,B 0.000,C 90.000,E1 240.411} C_DIS
LIN {X -0.146,Y -502.256,Z 1040.127,A 0.000,B 0.000,C 90.000,E1 238.948} C_DIS
LIN {X 0.095,Y -498.908,Z 1040.117,A 0.000,B 0.000,C 90.000,E1 237.120} C_DIS
LIN {X -0.017,Y -496.544,Z 1040.111,A 0.000,B 0.000,C 90.000,E1 235.928} C_DIS
LIN {X -0.038,Y -492.622,Z 1040.101,A 0.000,B 0.000,C 90.000,E1 234.116} C_DIS
LIN {X 0.289,Y -489.111,Z 1040.092,A 0.000,B 0.000,C 90.000,E1 232.557} C_DIS
LIN {X -0.071,Y -483.394,Z 1040.079,A 0.000,B 0.000,C 90.000,E1 230.150} C_DIS
LIN {X -0.027,Y -478.008,Z 1040.065,A 0.000,B 0.000,C 90.000,E1 227.676} C_DIS
LIN {X -0.119,Y -474.828,Z 1040.056,A 0.000,B 0.000,C 90.000,E1 226.134} C_DIS
LIN {X -0.196,Y -470.958,Z 1040.046,A 0.000,B 0.000,C 90.000,E1 224.271} C_DIS
LIN {X 0.043,Y -466.439,Z 1040.034,A 0.000,B 0.000,C 90.000,E1 222.043} C_DIS
LIN {X 0.079,Y -463.251,Z 1040.025,A 0.000,B 0.000,C 90.000,E1 220.458} C_DIS
LIN {X -0.239,Y -459.897,Z 1040.016,A 0.000,B 0.000,C 90.000,E1 218.910} C_DIS
LIN {X 0.022,Y -456.439,Z 1040.007,A 0.000,B 0.000,C 90.000,E1 217.282} C_DIS
LIN {X -0.062,Y -453.629,Z 1040.000,A 0.000,B 0.000,C 90.000,E1 216.011} C_DIS
LIN {X 0.183,Y -451.041,Z 1039.993,A 0.000,B 0.000,C 90.000,E1 214.692} C_DIS
LIN {X -0.143,Y -446.295,Z 1039.980,A 0.000,B 0.000,C 90.000,E1 212.467} C_DIS
LIN {X 0.231,Y -441.978,Z 1039.969,A 0.000,B 0.000,C 90.000,E1 210.463} C_DIS
LIN {X -0.141,Y -438.286,Z 1039.960,A 0.000,B 0.000,C 90.000,E1 208.871} C_DIS
LIN {X -0.175,Y -432.355,Z 1039.946,A 0.000,B 0.000,C 90.000,E1 206.232} C_DIS
LIN {X 0.192,Y -426.624,Z 1039.931,A 0.000,B 0.000,C 90.000,E1 203.515} C_DIS
LIN {X 0.029,Y -421.405,Z 1039.916,A 0.000,B 0.000,C 90.000,E1 200.844} C_DIS
LIN {X -0.091,Y -414.480,Z 1039.891,A 0.000,B 0.000,C 90.000,E1 196.441} C_DIS
LIN {X 0.128,Y -412.365,Z 1039.880,A 0.000,B 0.000,C 90.000,E1 194.356} C_DIS
LIN {X -0.055,Y -411.663,Z 1039.872,A 0.000,B 0.000,C 90.000,E1 193.008} C_DIS
LIN {X 0.097,Y -411.573,Z 1039.868,A 0.000,B 0.000,C 90.000,E1 192.299} C_DIS
LIN {X -0.175,Y -411.751,Z 1039.867,A 0.000,B 0.000,C 90.000,E1 192.007} C_DIS
LIN {X -0.028,Y -412.589,Z 1039.863,A 0.000,B 0.000,C 90.000,E1 191.299} C_DIS
LIN {X 0.120,Y -414.189,Z 1039.859,A 0.000,B 0.000,C 90.000,E1 190.602} C_DIS
LIN {X -0.201,Y -416.906,Z 1039.855,A 0.000,B 0.000,C 90.000,E1 189.962} C_DIS
LIN {X -0.149,Y -418.460,Z 1039.853,A 0.000,B 0.000,C 90.000,E1 189.613} C_DIS
LIN {X 0.127,Y -423.166,Z 1039.849,A 0.000,B 0.000,C 90.000,E1 188.803} C_DIS
LIN {X -0.057,Y -438.704,Z 1039.837,A 0.000,B 0.000,C 90.000,E1 186.663} C_DIS
LIN {X 0.091,Y -443.326,Z 1039.834,A 0.000,B 0.000,C 90.000,E1 186.030} C_DIS
LIN {X -0.193,Y -444.595,Z 1039.833,A 0.000,B 0.000,C 90.000,E1 185.910} C_DIS
LIN {X 0.084,Y -447.984,Z 1039.830,A 0.000,B 0.000,C 90.000,E1 185.391} C_DIS
LIN {X -0.158,Y -451.694,Z 1039.827,A 0.000,B 0.000,C 90.000,E1 184.935} C_DIS
LIN {X 0.016,Y -457.511,Z 1039.823,A 0.000,B 0.000,C 90.000,E1 184.131} C_DIS
LIN {X 0.061,Y -463.302,Z 1039.819,A 0.000,B 0.000,C 90.000,E1 183.326} C_DIS
LIN {X -0.214,Y -468.763,Z 1039.814,A 0.000,B 0.000,C 90.000,E1 182.579} C_DIS
LIN {X -0.065,Y -474.256,Z 1039.810,A 0.000,B 0.000,C 90.000,E1 181.776} C_DIS
LIN {X -0.006,Y -478.337,Z 1039.806,A 0.000,B 0.000,C 90.000,E1 181.146} C_DIS
LIN {X 0.098,Y -482.417,Z 1039.803,A 0.000,B 0.000,C 90.000,E1 180.516} C_DIS
LIN {X 0.074,Y -488.341,Z 1039.798,A 0.000,B 0.000,C 90.000,E1 179.599} C_DIS
LIN {X 0.083,Y -494.167,Z 1039.793,A 0.000,B 0.000,C 90.000,E1 178.682} C_DIS
LIN {X 0.171,Y -499.875,Z 1039.788,A 0.000,B 0.000,C 90.000,E1 177.764} C_DIS
LIN {X 0.220,Y -507.003,Z 1039.781,A 0.000,B 0.000,C 90.000,E1 176.560} C_DIS
LIN {X -0.186,Y -515.593,Z 1039.773,A 0.000,B 0.000,C 90.000,E1 175.122} C_DIS
LIN {X 0.075,Y -524.061,Z 1039.765,A 0.000,B 0.000,C 90.000,E1 173.628} C_DIS
LIN {X 0.021,Y -532.311,Z 1039.757,A 0.000,B 0.000,C 90.000,E1 172.186} C_DIS
LIN {X 0.072,Y -537.098,Z 1039.752,A 0.000,B 0.000,C 90.000,E1 171.319} C_DIS
LIN {X -0.196,Y -543.430,Z 1039.745,A 0.000,B 0.000,C 90.000,E1 170.208} C_DIS
LIN {X 0.017,Y -551.968,Z 1039.737,A 0.000,B 0.000,C 90.000,E1 168.634} C_DIS
LIN {X 0.113,Y -559.495,Z 1039.729,A 0.000,B 0.000,C 90.000,E1 167.229} C_DIS
LIN {X -0.116,Y -564.557,Z 1039.724,A 0.000,B 0.000,C 90.000,E1 166.284} C_DIS
LIN {X -0.108,Y -570.858,Z 1039.717,A 0.000,B 0.000,C 90.000,E1 165.046} C_DIS
LIN {X 0.246,Y -576.249,Z 1039.711,A 0.000,B 0.000,C 90.000,E1 163.921} C_DIS
LIN {X 0.116,Y -581.416,Z 1039.705,A 0.000,B 0.000,C 90.000,E1 162.851} C_DIS
LIN {X 0.227,Y -586.254,Z 1039.699,A 0.000,B 0.000,C 90.000,E1 161.764} C_DIS
LIN {X -0.158,Y -590.829,Z 1039.693,A 0.000,B 0.000,C 90.000,E1 160.732} C_DIS
LIN {X 0.074,Y -595.091,Z 1039.687,A 0.000,B 0.000,C 90.000,E1 159.645} C_DIS
LIN {X 0.014,Y -599.035,Z 1039.681,A 0.000,B 0.000,C 90.000,E1 158.592} C_DIS
LIN {X -0.056,Y -603.624,Z 1039.674,A 0.000,B 0.000,C 90.000,E1 157.283} C_DIS
LIN {X 0.009,Y -607.088,Z 1039.668,A 0.000,B 0.000,C 90.000,E1 156.230} C_DIS
LIN {X 0.113,Y -610.336,Z 1039.662,A 0.000,B 0.000,C 90.000,E1 155.177} C_DIS
LIN {X -0.071,Y -614.015,Z 1039.655,A 0.000,B 0.000,C 90.000,E1 153.896} C_DIS
LIN {X -0.190,Y -617.468,Z 1039.648,A 0.000,B 0.000,C 90.000,E1 152.615} C_DIS
LIN {X -0.237,Y -619.499,Z 1039.644,A 0.000,B 0.000,C 90.000,E1 151.847} C_DIS
LIN {X 0.322,Y -623.969,Z 1039.634,A 0.000,B 0.000,C 90.000,E1 149.999} C_DIS
LIN {X 0.122,Y -627.689,Z 1039.625,A 0.000,B 0.000,C 90.000,E1 148.486} C_DIS
LIN {X 0.287,Y -630.060,Z 1039.619,A 0.000,B 0.000,C 90.000,E1 147.454} C_DIS
LIN {X -0.008,Y -633.596,Z 1039.611,A 0.000,B 0.000,C 90.000,E1 145.960} C_DIS
LIN {X -0.406,Y -637.018,Z 1039.603,A 0.000,B 0.000,C 90.000,E1 144.482} C_DIS
LIN {X 0.259,Y -639.319,Z 1039.597,A 0.000,B 0.000,C 90.000,E1 143.417} C_DIS
LIN {X -0.134,Y -643.360,Z 1039.587,A 0.000,B 0.000,C 90.000,E1 141.698} C_DIS
LIN {X 0.365,Y -647.346,Z 1039.578,A 0.000,B 0.000,C 90.000,E1 139.908} C_DIS
LIN {X -0.449,Y -651.308,Z 1039.568,A 0.000,B 0.000,C 90.000,E1 138.243} C_DIS
LIN {X 0.103,Y -656.620,Z 1039.556,A 0.000,B 0.000,C 90.000,E1 135.972} C_DIS
LIN {X -0.169,Y -664.554,Z 1039.539,A 0.000,B 0.000,C 90.000,E1 133.056} C_DIS
LIN {X -0.165,Y -669.359,Z 1039.530,A 0.000,B 0.000,C 90.000,E1 131.353} C_DIS
LIN {X -0.082,Y -672.752,Z 1039.523,A 0.000,B 0.000,C 90.000,E1 130.135} C_DIS
LIN {X 0.147,Y -676.130,Z 1039.516,A 0.000,B 0.000,C 90.000,E1 128.910} C_DIS
LIN {X -0.104,Y -678.677,Z 1039.511,A 0.000,B 0.000,C 90.000,E1 127.971} C_DIS
LIN {X 0.260,Y -682.358,Z 1039.503,A 0.000,B 0.000,C 90.000,E1 126.503} C_DIS
LIN {X -0.122,Y -686.079,Z 1039.495,A 0.000,B 0.000,C 90.000,E1 125.105} C_DIS
LIN {X 0.138,Y -689.694,Z 1039.487,A 0.000,B 0.000,C 90.000,E1 123.658} C_DIS
LIN {X -0.116,Y -693.185,Z 1039.479,A 0.000,B 0.000,C 90.000,E1 122.260} C_DIS
LIN {X 0.247,Y -695.913,Z 1039.473,A 0.000,B 0.000,C 90.000,E1 121.052} C_DIS
LIN {X 0.046,Y -697.865,Z 1039.467,A 0.000,B 0.000,C 90.000,E1 120.129} C_DIS
LIN {X 0.217,Y -699.024,Z 1039.464,A 0.000,B 0.000,C 90.000,E1 119.411} C_DIS
LIN {X 0.327,Y -700.568,Z 1039.457,A 0.000,B 0.000,C 90.000,E1 118.231} C_DIS
LIN {X -0.216,Y -702.173,Z 1039.449,A 0.000,B 0.000,C 90.000,E1 116.873} C_DIS
LIN {X -0.008,Y -702.888,Z 1039.445,A 0.000,B 0.000,C 90.000,E1 116.155} C_DIS
LIN {X 0.176,Y -703.661,Z 1039.440,A 0.000,B 0.000,C 90.000,E1 115.207} C_DIS
LIN {X -0.194,Y -703.964,Z 1039.438,A 0.000,B 0.000,C 90.000,E1 114.771} C_DIS
LIN {X 0.082,Y -703.911,Z 1039.435,A 0.000,B 0.000,C 90.000,E1 114.283} C_DIS
LIN {X -0.276,Y -703.790,Z 1039.434,A 0.000,B 0.000,C 90.000,E1 114.079} C_DIS
LIN {X 0.003,Y -702.779,Z 1039.431,A 0.000,B 0.000,C 90.000,E1 113.590} C_DIS
LIN {X 0.282,Y -702.045,Z 1039.430,A 0.000,B 0.000,C 90.000,E1 113.334} C_DIS
LIN {X -0.092,Y -699.247,Z 1039.427,A 0.000,B 0.000,C 90.000,E1 112.898} C_DIS
LIN {X 0.041,Y -698.445,Z 1039.427,A 0.000,B 0.000,C 90.000,E1 112.770} C_DIS
LIN {X 0.172,Y -697.273,Z 1039.426,A 0.000,B 0.000,C 90.000,E1 112.642} C_DIS
LIN {X 0.303,Y -695.469,Z 1039.425,A 0.000,B 0.000,C 90.000,E1 112.514} C_DIS
LIN {X -0.031,Y -690.216,Z 1039.424,A 0.000,B 0.000,C 90.000,E1 112.259} C_DIS
LIN {X 0.252,Y -688.526,Z 1039.423,A 0.000,B 0.000,C 90.000,E1 112.153} C_DIS
LIN {X 0.156,Y -686.088,Z 1039.423,A 0.000,B 0.000,C 90.000,E1 112.078} C_DIS
LIN {X 0.099,Y -684.002,Z 1039.422,A 0.000,B 0.000,C 90.000,E1 112.025} C_DIS
LIN {X 0.397,Y -675.352,Z 1039.422,A 0.000,B 0.000,C 90.000,E1 111.897} C_DIS
LIN {X 0.306,Y -611.497,Z 1039.422,A 0.000,B 0.000,C 90.000,E1 111.897} C_DIS
LIN {X -0.020,Y -605.200,Z 1039.421,A 0.000,B 0.000,C 90.000,E1 111.716} C_DIS
LIN {X -0.058,Y -602.292,Z 1039.420,A 0.000,B 0.000,C 90.000,E1 111.589} C_DIS
LIN {X -0.175,Y -597.545,Z 1039.419,A 0.000,B 0.000,C 90.000,E1 111.354} C_DIS
LIN {X -0.117,Y -591.858,Z 1039.417,A 0.000,B 0.000,C 90.000,E1 110.972} C_DIS
LIN {X -0.063,Y -585.005,Z 1039.413,A 0.000,B 0.000,C 90.000,E1 110.429} C_DIS
LIN {X 0.154,Y -576.696,Z 1039.410,A 0.000,B 0.000,C 90.000,E1 109.704} C_DIS
LIN {X -0.037,Y -570.540,Z 1039.407,A 0.000,B 0.000,C 90.000,E1 109.268} C_DIS
LIN {X -0.070,Y -565.458,Z 1039.405,A 0.000,B 0.000,C 90.000,E1 108.960} C_DIS
LIN {X -0.002,Y -560.507,Z 1039.404,A 0.000,B 0.000,C 90.000,E1 108.671} C_DIS
LIN {X 0.142,Y -554.140,Z 1039.402,A 0.000,B 0.000,C 90.000,E1 108.308} C_DIS
LIN {X -0.235,Y -549.547,Z 1039.400,A 0.000,B 0.000,C 90.000,E1 108.055} C_DIS
LIN {X 0.121,Y -547.966,Z 1039.399,A 0.000,B 0.000,C 90.000,E1 107.819} C_DIS
LIN {X 0.079,Y -547.959,Z 1039.399,A 0.000,B 0.000,C 90.000,E1 107.819} C_DIS
LIN {X -0.228,Y -547.502,Z 1039.398,A 0.000,B 0.000,C 90.000,E1 107.583} C_DIS
LIN {X -0.097,Y -547.577,Z 1039.394,A 0.000,B 0.000,C 90.000,E1 106.985} C_DIS
LIN {X -0.040,Y -548.159,Z 1039.390,A 0.000,B 0.000,C 90.000,E1 106.134} C_DIS
LIN {X -0.028,Y -549.396,Z 1039.377,A 0.000,B 0.000,C 90.000,E1 103.883} C_DIS
LIN {X 0.242,Y -552.202,Z 1039.359,A 0.000,B 0.000,C 90.000,E1 100.489} C_DIS
LIN {X 0.066,Y -554.955,Z 1039.344,A 0.000,B 0.000,C 90.000,E1 97.992} C_DIS
LIN {X -0.004,Y -556.554,Z 1039.337,A 0.000,B 0.000,C 90.000,E1 96.606} C_DIS
LIN {X -0.051,Y -558.005,Z 1039.329,A 0.000,B 0.000,C 90.000,E1 95.220} C_DIS
LIN {X -0.253,Y -558.854,Z 1039.323,A 0.000,B 0.000,C 90.000,E1 94.131} C_DIS
LIN {X 0.035,Y -559.476,Z 1039.318,A 0.000,B 0.000,C 90.000,E1 93.269} C_DIS
LIN {X 0.060,Y -560.284,Z 1039.309,A 0.000,B 0.000,C 90.000,E1 91.604} C_DIS
LIN {X 0.063,Y -560.882,Z 1039.300,A 0.000,B 0.000,C 90.000,E1 89.943} C_DIS
LIN {X 0.194,Y -561.540,Z 1039.289,A 0.000,B 0.000,C 90.000,E1 87.993} C_DIS
LIN {X 0.239,Y -562.080,Z 1039.280,A 0.000,B 0.000,C 90.000,E1 86.331} C_DIS
LIN {X 0.230,Y -562.549,Z 1039.272,A 0.000,B 0.000,C 90.000,E1 84.951} C_DIS
LIN {X 0.226,Y -562.881,Z 1039.264,A 0.000,B 0.000,C 90.000,E1 83.571} C_DIS
LIN {X 0.114,Y -563.427,Z 1039.252,A 0.000,B 0.000,C 90.000,E1 81.376} C_DIS
LIN {X -0.191,Y -564.329,Z 1039.238,A 0.000,B 0.000,C 90.000,E1 78.926} C_DIS
LIN {X -0.128,Y -565.230,Z 1039.228,A 0.000,B 0.000,C 90.000,E1 76.992} C_DIS
LIN {X 0.084,Y -566.420,Z 1039.217,A 0.000,B 0.000,C 90.000,E1 75.046} C_DIS
LIN {X 0.082,Y -568.062,Z 1039.205,A 0.000,B 0.000,C 90.000,E1 72.851} C_DIS
LIN {X -0.013,Y -568.973,Z 1039.199,A 0.000,B 0.000,C 90.000,E1 71.764} C_DIS
LIN {X 0.065,Y -570.289,Z 1039.190,A 0.000,B 0.000,C 90.000,E1 70.115} C_DIS
LIN {X 0.001,Y -571.051,Z 1039.184,A 0.000,B 0.000,C 90.000,E1 69.028} C_DIS
LIN {X -0.028,Y -572.059,Z 1039.176,A 0.000,B 0.000,C 90.000,E1 67.667} C_DIS
LIN {X -0.208,Y -573.051,Z 1039.167,A 0.000,B 0.000,C 90.000,E1 66.049} C_DIS
LIN {X -0.136,Y -573.951,Z 1039.158,A 0.000,B 0.000,C 90.000,E1 64.409} C_DIS
LIN {X 0.204,Y -574.765,Z 1039.149,A 0.000,B 0.000,C 90.000,E1 62.743} C_DIS
LIN {X 0.202,Y -575.341,Z 1039.141,A 0.000,B 0.000,C 90.000,E1 61.385} C_DIS
LIN {X -0.324,Y -576.112,Z 1039.131,A 0.000,B 0.000,C 90.000,E1 59.537} C_DIS
LIN {X 0.129,Y -576.524,Z 1039.125,A 0.000,B 0.000,C 90.000,E1 58.408} C_DIS
LIN {X 0.242,Y -576.984,Z 1039.117,A 0.000,B 0.000,C 90.000,E1 57.041} C_DIS
LIN {X -0.268,Y -577.270,Z 1039.111,A 0.000,B 0.000,C 90.000,E1 56.008} C_DIS
LIN {X 0.028,Y -577.477,Z 1039.105,A 0.000,B 0.000,C 90.000,E1 54.895} C_DIS
LIN {X 0.016,Y -577.589,Z 1039.098,A 0.000,B 0.000,C 90.000,E1 53.543} C_DIS
LIN {X 0.146,Y -577.567,Z 1039.093,A 0.000,B 0.000,C 90.000,E1 52.718} C_DIS
LIN {X 0.005,Y -577.523,Z 1039.090,A 0.000,B 0.000,C 90.000,E1 52.190} C_DIS
LIN {X 0.027,Y -577.328,Z 1039.085,A 0.000,B 0.000,C 90.000,E1 51.376} C_DIS
LIN {X 0.065,Y -576.559,Z 1039.076,A 0.000,B 0.000,C 90.000,E1 49.747} C_DIS
LIN {X -0.069,Y -575.798,Z 1039.069,A 0.000,B 0.000,C 90.000,E1 48.405} C_DIS
LIN {X -0.266,Y -574.733,Z 1039.061,A 0.000,B 0.000,C 90.000,E1 47.067} C_DIS
LIN {X 0.100,Y -573.980,Z 1039.057,A 0.000,B 0.000,C 90.000,E1 46.215} C_DIS
LIN {X 0.334,Y -573.409,Z 1039.054,A 0.000,B 0.000,C 90.000,E1 45.648} C_DIS
LIN {X -0.022,Y -571.879,Z 1039.048,A 0.000,B 0.000,C 90.000,E1 44.595} C_DIS
LIN {X -0.100,Y -570.607,Z 1039.043,A 0.000,B 0.000,C 90.000,E1 43.785} C_DIS
LIN {X -0.083,Y -568.707,Z 1039.037,A 0.000,B 0.000,C 90.000,E1 42.690} C_DIS
LIN {X 0.217,Y -567.078,Z 1039.033,A 0.000,B 0.000,C 90.000,E1 41.838} C_DIS
LIN {X -0.302,Y -565.175,Z 1039.028,A 0.000,B 0.000,C 90.000,E1 41.067} C_DIS
LIN {X -0.046,Y -563.090,Z 1039.023,A 0.000,B 0.000,C 90.000,E1 40.216} C_DIS
LIN {X 0.156,Y -561.576,Z 1039.020,A 0.000,B 0.000,C 90.000,E1 39.644} C_DIS
LIN {X 0.011,Y -559.034,Z 1039.016,A 0.000,B 0.000,C 90.000,E1 38.830} C_DIS
LIN {X -0.162,Y -556.246,Z 1039.011,A 0.000,B 0.000,C 90.000,E1 38.016} C_DIS
LIN {X 0.074,Y -553.060,Z 1039.006,A 0.000,B 0.000,C 90.000,E1 37.156} C_DIS
LIN {X 0.212,Y -550.824,Z 1039.003,A 0.000,B 0.000,C 90.000,E1 36.583} C_DIS
LIN {X 0.065,Y -547.097,Z 1038.999,A 0.000,B 0.000,C 90.000,E1 35.758} C_DIS
LIN {X 0.331,Y -543.718,Z 1038.995,A 0.000,B 0.000,C 90.000,E1 35.025} C_DIS
LIN {X 0.107,Y -539.426,Z 1038.990,A 0.000,B 0.000,C 90.000,E1 34.199} C_DIS
LIN {X -0.161,Y -533.266,Z 1038.984,A 0.000,B 0.000,C 90.000,E1 33.086} C_DIS
LIN {X 0.109,Y -529.082,Z 1038.980,A 0.000,B 0.000,C 90.000,E1 32.339} C_DIS
LIN {X 0.016,Y -522.751,Z 1038.974,A 0.000,B 0.000,C 90.000,E1 31.337} C_DIS
LIN {X 0.014,Y -516.767,Z 1038.969,A 0.000,B 0.000,C 90.000,E1 30.463} C_DIS
LIN {X 0.038,Y -512.476,Z 1038.966,A 0.000,B 0.000,C 90.000,E1 29.873} C_DIS
LIN {X 0.210,Y -509.110,Z 1038.964,A 0.000,B 0.000,C 90.000,E1 29.411} C_DIS
LIN {X 0.177,Y -504.307,Z 1038.960,A 0.000,B 0.000,C 90.000,E1 28.821} C_DIS
LIN {X -0.138,Y -500.402,Z 1038.958,A 0.000,B 0.000,C 90.000,E1 28.409} C_DIS
LIN {X 0.152,Y -493.678,Z 1038.954,A 0.000,B 0.000,C 90.000,E1 27.641} C_DIS
LIN {X -0.061,Y -486.775,Z 1038.950,A 0.000,B 0.000,C 90.000,E1 26.950} C_DIS
LIN {X -0.042,Y -476.843,Z 1038.944,A 0.000,B 0.000,C 90.000,E1 25.976} C_DIS
LIN {X -0.002,Y -466.680,Z 1038.939,A 0.000,B 0.000,C 90.000,E1 25.027} C_DIS
LIN {X 0.218,Y -457.596,Z 1038.935,A 0.000,B 0.000,C 90.000,E1 24.207} C_DIS
LIN {X 0.029,Y -444.016,Z 1038.928,A 0.000,B 0.000,C 90.000,E1 23.078} C_DIS
LIN {X 0.250,Y -424.595,Z 1038.918,A 0.000,B 0.000,C 90.000,E1 21.280} C_DIS
LIN {X 0.077,Y -413.064,Z 1038.912,A 0.000,B 0.000,C 90.000,E1 20.120} C_DIS
LIN {X 0.038,Y -401.832,Z 1038.905,A 0.000,B 0.000,C 90.000,E1 18.852} C_DIS
LIN {X -0.060,Y -397.082,Z 1038.901,A 0.000,B 0.000,C 90.000,E1 18.236} C_DIS
LIN {X 0.015,Y -394.284,Z 1038.899,A 0.000,B 0.000,C 90.000,E1 17.764} C_DIS
LIN {X 0.151,Y -393.577,Z 1038.898,A 0.000,B 0.000,C 90.000,E1 17.583} C_DIS
LIN {X 0.039,Y -391.881,Z 1038.895,A 0.000,B 0.000,C 90.000,E1 17.040} C_DIS
LIN {X -0.044,Y -391.285,Z 1038.891,A 0.000,B 0.000,C 90.000,E1 16.386} C_DIS
LIN {X -0.080,Y -391.413,Z 1038.888,A 0.000,B 0.000,C 90.000,E1 15.843} C_DIS
LIN {X -0.142,Y -397.349,Z 1038.860,A 0.000,B 0.000,C 90.000,E1 10.894} C_DIS
LIN {X 0.087,Y -403.958,Z 1038.839,A 0.000,B 0.000,C 90.000,E1 7.004} C_DIS
LIN {X -0.016,Y -409.088,Z 1038.826,A 0.000,B 0.000,C 90.000,E1 4.588} C_DIS
LIN {X -0.045,Y -412.187,Z 1038.818,A 0.000,B 0.000,C 90.000,E1 3.212} C_DIS
LIN {X 0.033,Y -413.901,Z 1038.815,A 0.000,B 0.000,C 90.000,E1 2.694} C_DIS
LIN {X 0.033,Y -414.669,Z 1038.814,A 0.000,B 0.000,C 90.000,E1 2.522} C_DIS
LIN {X -0.092,Y -417.339,Z 1038.811,A 0.000,B 0.000,C 90.000,E1 2.064} C_DIS
LIN {X 0.120,Y -417.930,Z 1038.811,A 0.000,B 0.000,C 90.000,E1 1.949} C_DIS
LIN {X -0.076,Y -422.696,Z 1038.808,A 0.000,B 0.000,C 90.000,E1 1.489} C_DIS
LIN {X -0.031,Y -429.730,Z 1038.806,A 0.000,B 0.000,C 90.000,E1 1.031} C_DIS
LIN {X 0.210,Y -442.876,Z 1038.801,A 0.000,B 0.000,C 90.000,E1 0.172} C_DIS
LIN {X -0.005,Y -461.062,Z 1038.795,A 0.000,B 0.000,C 90.000,E1 359.083} C_DIS
LIN {X 0.033,Y -474.296,Z 1038.791,A 0.000,B 0.000,C 90.000,E1 358.282} C_DIS
LIN {X -0.243,Y -489.012,Z 1038.786,A 0.000,B 0.000,C 90.000,E1 357.421} C_DIS
LIN {X -0.076,Y -497.027,Z 1038.783,A 0.000,B 0.000,C 90.000,E1 356.906} C_DIS
LIN {X -0.013,Y -504.877,Z 1038.780,A 0.000,B 0.000,C 90.000,E1 356.388} C_DIS
LIN {X -0.210,Y -514.259,Z 1038.776,A 0.000,B 0.000,C 90.000,E1 355.755} C_DIS
LIN {X -0.133,Y -518.664,Z 1038.775,A 0.000,B 0.000,C 90.000,E1 355.412} C_DIS
LIN {X -0.070,Y -524.458,Z 1038.772,A 0.000,B 0.000,C 90.000,E1 354.951} C_DIS
LIN {X 0.209,Y -531.551,Z 1038.769,A 0.000,B 0.000,C 90.000,E1 354.318} C_DIS
LIN {X 0.127,Y -538.350,Z 1038.765,A 0.000,B 0.000,C 90.000,E1 353.685} C_DIS
LIN {X 0.006,Y -543.569,Z 1038.762,A 0.000,B 0.000,C 90.000,E1 353.166} C_DIS
LIN {X 0.277,Y -549.551,Z 1038.758,A 0.000,B 0.000,C 90.000,E1 352.470} C_DIS
LIN {X 0.160,Y -555.098,Z 1038.755,A 0.000,B 0.000,C 90.000,E1 351.781} C_DIS
LIN {X -0.138,Y -559.138,Z 1038.751,A 0.000,B 0.000,C 90.000,E1 351.254} C_DIS
LIN {X -0.095,Y -563.669,Z 1038.748,A 0.000,B 0.000,C 90.000,E1 350.557} C_DIS
LIN {X -0.010,Y -567.785,Z 1038.744,A 0.000,B 0.000,C 90.000,E1 349.859} C_DIS
LIN {X -0.315,Y -570.876,Z 1038.741,A 0.000,B 0.000,C 90.000,E1 349.342} C_DIS
LIN {X 0.263,Y -575.224,Z 1038.736,A 0.000,B 0.000,C 90.000,E1 348.465} C_DIS
LIN {X -0.238,Y -579.171,Z 1038.732,A 0.000,B 0.000,C 90.000,E1 347.701} C_DIS
LIN {X 0.100,Y -582.163,Z 1038.728,A 0.000,B 0.000,C 90.000,E1 346.992} C_DIS
LIN {X -0.096,Y -586.710,Z 1038.722,A 0.000,B 0.000,C 90.000,E1 345.936} C_DIS
LIN {X -0.088,Y -591.093,Z 1038.716,A 0.000,B 0.000,C 90.000,E1 344.866} C_DIS
LIN {X 0.253,Y -596.252,Z 1038.708,A 0.000,B 0.000,C 90.000,E1 343.504} C_DIS
LIN {X 0.279,Y -601.118,Z 1038.701,A 0.000,B 0.000,C 90.000,E1 342.181} C_DIS
LIN {X 0.095,Y -604.757,Z 1038.695,A 0.000,B 0.000,C 90.000,E1 341.148} C_DIS
LIN {X -0.313,Y -608.875,Z 1038.688,A 0.000,B 0.000,C 90.000,E1 339.880} C_DIS
LIN {X 0.120,Y -612.578,Z 1038.681,A 0.000,B 0.000,C 90.000,E1 338.539} C_DIS
LIN {X -0.265,Y -615.341,Z 1038.675,A 0.000,B 0.000,C 90.000,E1 337.539} C_DIS
